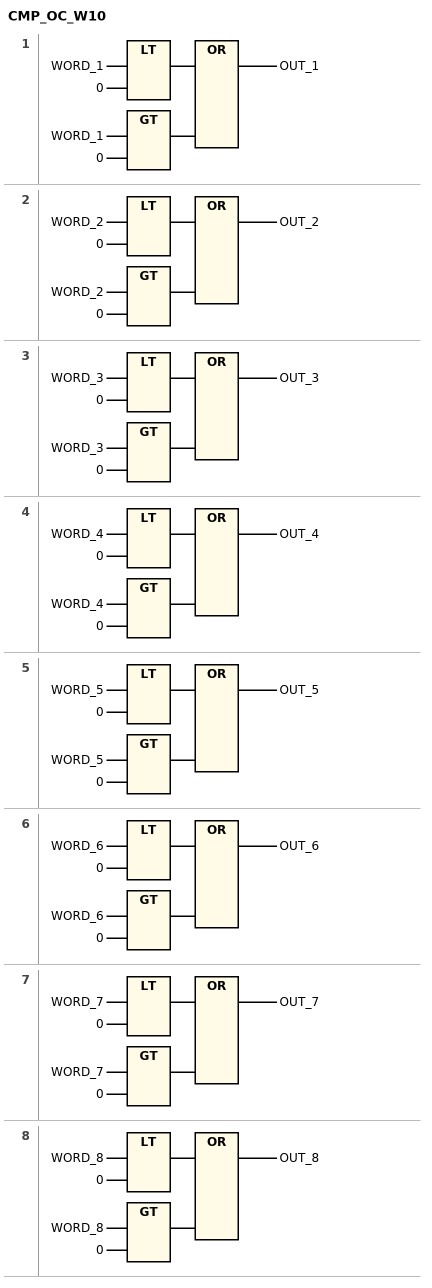
// NETWORK 1
OUT_1 := WORD_1 < 0 OR WORD_1 > 0;

// NETWORK 2
OUT_2 := WORD_2 < 0 OR WORD_2 > 0;

// NETWORK 3
OUT_3 := WORD_3 < 0 OR WORD_3 > 0;

// NETWORK 4
OUT_4 := WORD_4 < 0 OR WORD_4 > 0;

// NETWORK 5
OUT_5 := WORD_5 < 0 OR WORD_5 > 0;

// NETWORK 6
OUT_6 := WORD_6 < 0 OR WORD_6 > 0;

// NETWORK 7
OUT_7 := WORD_7 < 0 OR WORD_7 > 0;

// NETWORK 8
OUT_8 := WORD_8 < 0 OR WORD_8 > 0;

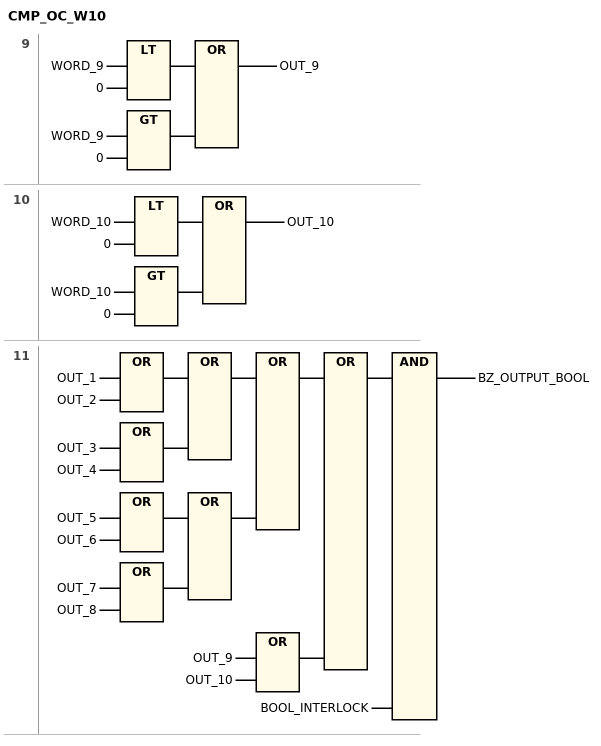
// NETWORK 9
OUT_9 := WORD_9 < 0 OR WORD_9 > 0;

// NETWORK 10
OUT_10 := WORD_10 < 0 OR WORD_10 > 0;

// NETWORK 11
BZ_OUTPUT_BOOL := ((((OUT_1 OR OUT_2) OR (OUT_3 OR OUT_4)) OR ((OUT_5 OR OUT_6) OR (OUT_7 OR OUT_8))) OR (OUT_9 OR OUT_10)) AND BOOL_INTERLOCK;

END_FUNCTION_BLOCK

// ---- FBs/B_JKS_OldFB/Word to Bit/CMP_OC_W2.TcPOU
FUNCTION_BLOCK CMP_OC_W2

VAR_INPUT
	BOOL_INTERLOCK : BOOL; (*INTERLOCK*)
	WORD_1: WORD;		(*WORD 1*)
	WORD_2: WORD;		(*WORD 2*)
	END_VAR


VAR_OUTPUT
	BZ_OUTPUT_BOOL : BOOL;
END_VAR


VAR
	OUT_1: BOOL;
	OUT_2: BOOL;
END_VAR

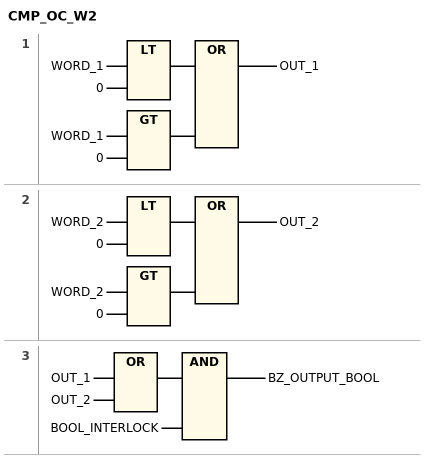
// NETWORK 1
OUT_1 := WORD_1 < 0 OR WORD_1 > 0;

// NETWORK 2
OUT_2 := WORD_2 < 0 OR WORD_2 > 0;

// NETWORK 3
BZ_OUTPUT_BOOL := (OUT_1 OR OUT_2) AND BOOL_INTERLOCK;

END_FUNCTION_BLOCK

// ---- FBs/B_JKS_OldFB/Word to Bit/CMP_OC_W3.TcPOU
FUNCTION_BLOCK CMP_OC_W3

VAR_INPUT
	BOOL_INTERLOCK : BOOL; (*INTERLOCK*)
	WORD_1: WORD;		(*WORD 1*)
	WORD_2: WORD;		(*WORD 2*)
	WORD_3: WORD;		(*WORD 3*)
	END_VAR


VAR_OUTPUT
	BZ_OUTPUT_BOOL : BOOL;
END_VAR


VAR
	OUT_1: BOOL;
	OUT_2: BOOL;
	OUT_3: BOOL;
END_VAR

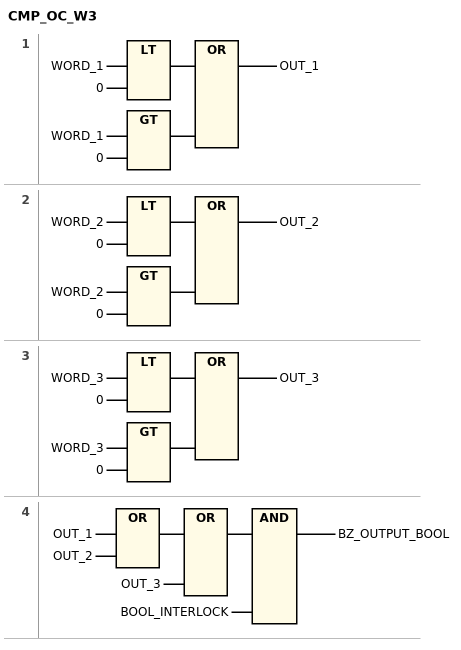
// NETWORK 1
OUT_1 := WORD_1 < 0 OR WORD_1 > 0;

// NETWORK 2
OUT_2 := WORD_2 < 0 OR WORD_2 > 0;

// NETWORK 3
OUT_3 := WORD_3 < 0 OR WORD_3 > 0;

// NETWORK 4
BZ_OUTPUT_BOOL := ((OUT_1 OR OUT_2) OR OUT_3) AND BOOL_INTERLOCK;

END_FUNCTION_BLOCK

// ---- FBs/B_JKS_OldFB/Word to Bit/CMP_OC_W4.TcPOU
FUNCTION_BLOCK CMP_OC_W4

VAR_INPUT
	BOOL_INTERLOCK : BOOL; (*INTERLOCK*)
	WORD_1: WORD;		(*WORD 1*)
	WORD_2: WORD;		(*WORD 2*)
	WORD_3: WORD;		(*WORD 3*)
	WORD_4: WORD;		(*WORD 4*)
	END_VAR


VAR_OUTPUT
	BZ_OUTPUT_BOOL : BOOL;
END_VAR


VAR
	OUT_1: BOOL;
	OUT_2: BOOL;
	OUT_3: BOOL;
	OUT_4: BOOL;
END_VAR

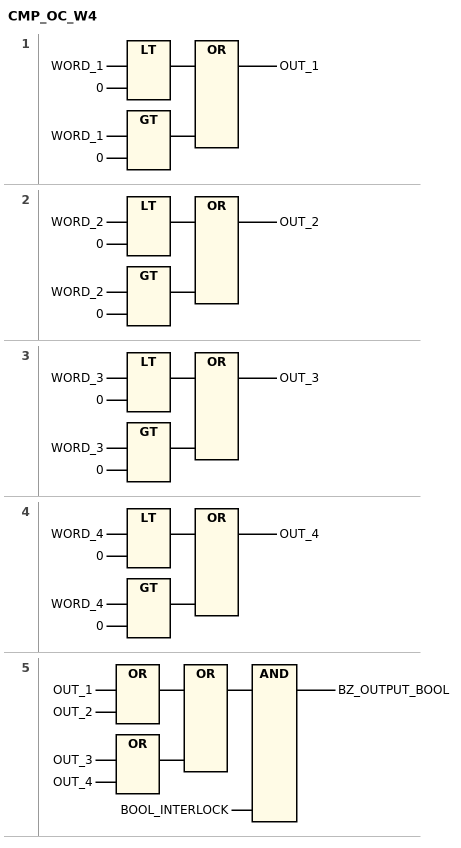
// NETWORK 1
OUT_1 := WORD_1 < 0 OR WORD_1 > 0;

// NETWORK 2
OUT_2 := WORD_2 < 0 OR WORD_2 > 0;

// NETWORK 3
OUT_3 := WORD_3 < 0 OR WORD_3 > 0;

// NETWORK 4
OUT_4 := WORD_4 < 0 OR WORD_4 > 0;

// NETWORK 5
BZ_OUTPUT_BOOL := ((OUT_1 OR OUT_2) OR (OUT_3 OR OUT_4)) AND BOOL_INTERLOCK;

END_FUNCTION_BLOCK

// ---- FBs/B_JKS_OldFB/Word to Bit/CMP_OC_W5.TcPOU
FUNCTION_BLOCK CMP_OC_W5

VAR_INPUT
	BOOL_INTERLOCK : BOOL; (*INTERLOCK*)
	WORD_1: WORD;		(*WORD 1*)
	WORD_2: WORD;		(*WORD 2*)
	WORD_3: WORD;		(*WORD 3*)
	WORD_4: WORD;		(*WORD 4*)
	WORD_5: WORD;		(*WORD 5*)
END_VAR


VAR_OUTPUT
	BZ_OUTPUT_BOOL : BOOL;
END_VAR


VAR
	OUT_1: BOOL;
	OUT_2: BOOL;
	OUT_3: BOOL;
	OUT_4: BOOL;
	OUT_5: BOOL;
END_VAR

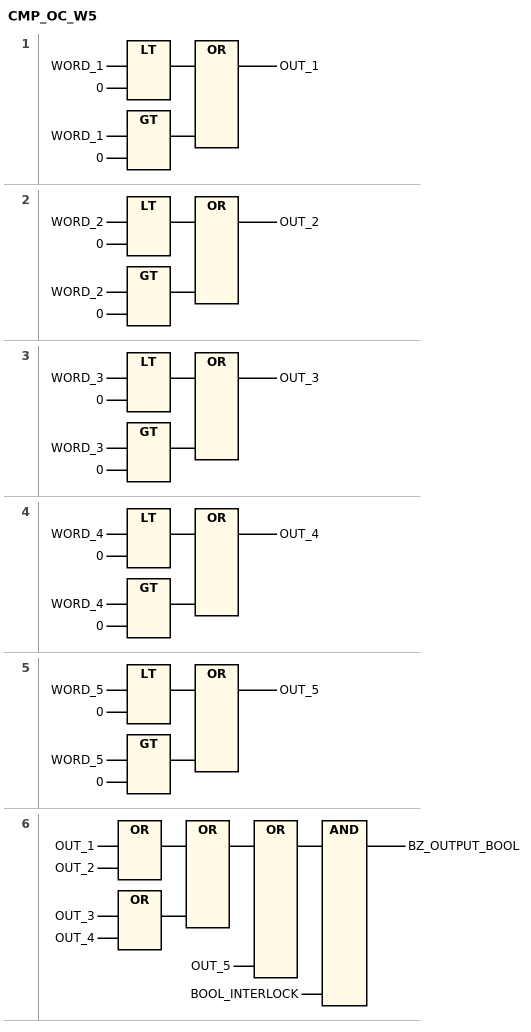
// NETWORK 1
OUT_1 := WORD_1 < 0 OR WORD_1 > 0;

// NETWORK 2
OUT_2 := WORD_2 < 0 OR WORD_2 > 0;

// NETWORK 3
OUT_3 := WORD_3 < 0 OR WORD_3 > 0;

// NETWORK 4
OUT_4 := WORD_4 < 0 OR WORD_4 > 0;

// NETWORK 5
OUT_5 := WORD_5 < 0 OR WORD_5 > 0;

// NETWORK 6
BZ_OUTPUT_BOOL := (((OUT_1 OR OUT_2) OR (OUT_3 OR OUT_4)) OR OUT_5) AND BOOL_INTERLOCK;

END_FUNCTION_BLOCK

// ---- FBs/B_JKS_OldFB/Word to Bit/CMP_OC_W6.TcPOU
FUNCTION_BLOCK CMP_OC_W6

VAR_INPUT
	BOOL_INTERLOCK : BOOL; (*INTERLOCK*)
	WORD_1: WORD;		(*WORD 1*)
	WORD_2: WORD;		(*WORD 2*)
	WORD_3: WORD;		(*WORD 3*)
	WORD_4: WORD;		(*WORD 4*)
	WORD_5: WORD;		(*WORD 5*)
	WORD_6: WORD;		(*WORD 6*)
END_VAR


VAR_OUTPUT
	BZ_OUTPUT_BOOL : BOOL;
END_VAR


VAR
	OUT_1: BOOL;
	OUT_2: BOOL;
	OUT_3: BOOL;
	OUT_4: BOOL;
	OUT_5: BOOL;
	OUT_6: BOOL;
END_VAR

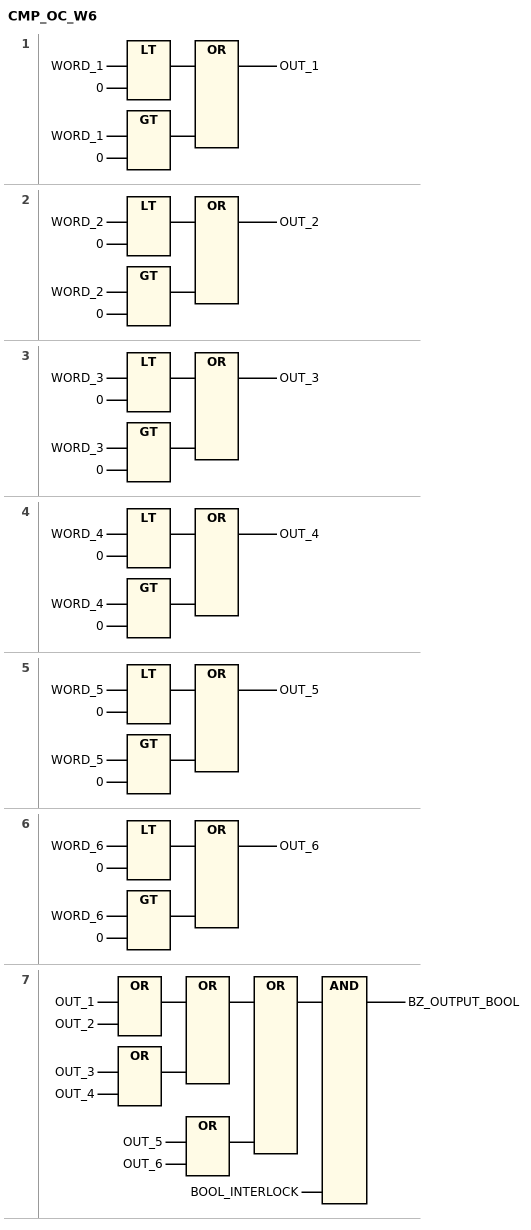
// NETWORK 1
OUT_1 := WORD_1 < 0 OR WORD_1 > 0;

// NETWORK 2
OUT_2 := WORD_2 < 0 OR WORD_2 > 0;

// NETWORK 3
OUT_3 := WORD_3 < 0 OR WORD_3 > 0;

// NETWORK 4
OUT_4 := WORD_4 < 0 OR WORD_4 > 0;

// NETWORK 5
OUT_5 := WORD_5 < 0 OR WORD_5 > 0;

// NETWORK 6
OUT_6 := WORD_6 < 0 OR WORD_6 > 0;

// NETWORK 7
BZ_OUTPUT_BOOL := (((OUT_1 OR OUT_2) OR (OUT_3 OR OUT_4)) OR (OUT_5 OR OUT_6)) AND BOOL_INTERLOCK;

END_FUNCTION_BLOCK

// ---- FBs/B_JKS_OldFB/Word to Bit/CMP_OC_W7.TcPOU
FUNCTION_BLOCK CMP_OC_W7

VAR_INPUT
	BOOL_INTERLOCK : BOOL; (*INTERLOCK*)
	WORD_1: WORD;		(*WORD 1*)
	WORD_2: WORD;		(*WORD 2*)
	WORD_3: WORD;		(*WORD 3*)
	WORD_4: WORD;		(*WORD 4*)
	WORD_5: WORD;		(*WORD 5*)
	WORD_6: WORD;		(*WORD 6*)
	WORD_7: WORD;		(*WORD 7*)
END_VAR


VAR_OUTPUT
	BZ_OUTPUT_BOOL : BOOL;
END_VAR


VAR
	OUT_1: BOOL;
	OUT_2: BOOL;
	OUT_3: BOOL;
	OUT_4: BOOL;
	OUT_5: BOOL;
	OUT_6: BOOL;
	OUT_7: BOOL;
END_VAR

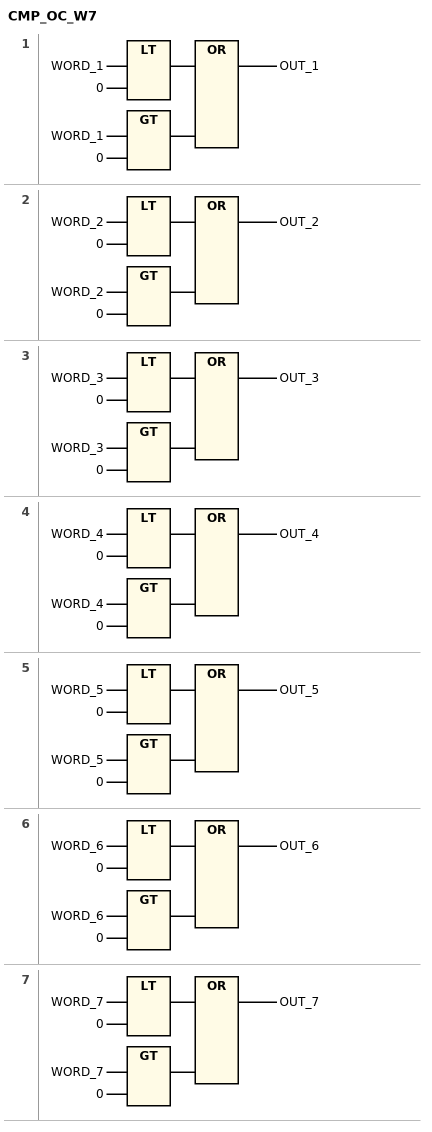
// NETWORK 1
OUT_1 := WORD_1 < 0 OR WORD_1 > 0;

// NETWORK 2
OUT_2 := WORD_2 < 0 OR WORD_2 > 0;

// NETWORK 3
OUT_3 := WORD_3 < 0 OR WORD_3 > 0;

// NETWORK 4
OUT_4 := WORD_4 < 0 OR WORD_4 > 0;

// NETWORK 5
OUT_5 := WORD_5 < 0 OR WORD_5 > 0;

// NETWORK 6
OUT_6 := WORD_6 < 0 OR WORD_6 > 0;

// NETWORK 7
OUT_7 := WORD_7 < 0 OR WORD_7 > 0;

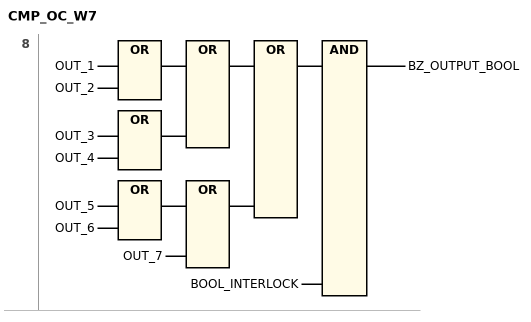
// NETWORK 8
BZ_OUTPUT_BOOL := (((OUT_1 OR OUT_2) OR (OUT_3 OR OUT_4)) OR ((OUT_5 OR OUT_6) OR OUT_7)) AND BOOL_INTERLOCK;

END_FUNCTION_BLOCK

// ---- FBs/B_JKS_OldFB/Word to Bit/CMP_OC_W8.TcPOU
FUNCTION_BLOCK CMP_OC_W8

VAR_INPUT
	BOOL_INTERLOCK : BOOL; (*INTERLOCK*)
	WORD_1: WORD;		(*WORD 1*)
	WORD_2: WORD;		(*WORD 2*)
	WORD_3: WORD;		(*WORD 3*)
	WORD_4: WORD;		(*WORD 4*)
	WORD_5: WORD;		(*WORD 5*)
	WORD_6: WORD;		(*WORD 6*)
	WORD_7: WORD;		(*WORD 7*)
	WORD_8: WORD;		(*WORD 8*)
END_VAR


VAR_OUTPUT
	BZ_OUTPUT_BOOL : BOOL;
END_VAR


VAR
	OUT_1: BOOL;
	OUT_2: BOOL;
	OUT_3: BOOL;
	OUT_4: BOOL;
	OUT_5: BOOL;
	OUT_6: BOOL;
	OUT_7: BOOL;
	OUT_8: BOOL;
END_VAR

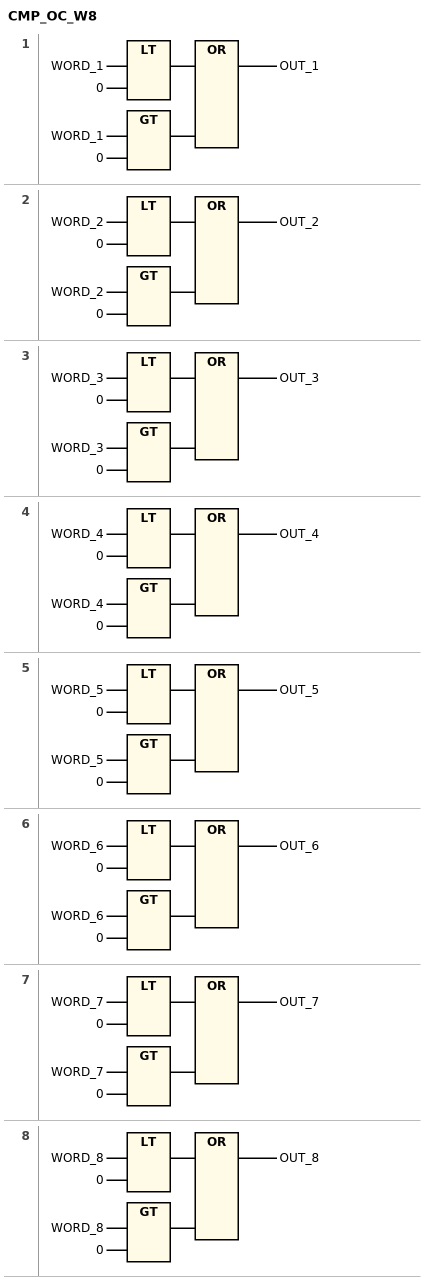
// NETWORK 1
OUT_1 := WORD_1 < 0 OR WORD_1 > 0;

// NETWORK 2
OUT_2 := WORD_2 < 0 OR WORD_2 > 0;

// NETWORK 3
OUT_3 := WORD_3 < 0 OR WORD_3 > 0;

// NETWORK 4
OUT_4 := WORD_4 < 0 OR WORD_4 > 0;

// NETWORK 5
OUT_5 := WORD_5 < 0 OR WORD_5 > 0;

// NETWORK 6
OUT_6 := WORD_6 < 0 OR WORD_6 > 0;

// NETWORK 7
OUT_7 := WORD_7 < 0 OR WORD_7 > 0;

// NETWORK 8
OUT_8 := WORD_8 < 0 OR WORD_8 > 0;

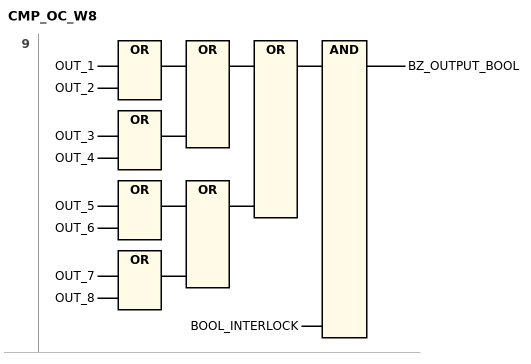
// NETWORK 9
BZ_OUTPUT_BOOL := (((OUT_1 OR OUT_2) OR (OUT_3 OR OUT_4)) OR ((OUT_5 OR OUT_6) OR (OUT_7 OR OUT_8))) AND BOOL_INTERLOCK;

END_FUNCTION_BLOCK

// ---- FBs/B_JKS_OldFB/Word to Bit/CMP_OC_W9.TcPOU
FUNCTION_BLOCK CMP_OC_W9

VAR_INPUT
	BOOL_INTERLOCK : BOOL; (*INTERLOCK*)
	WORD_1: WORD;		(*WORD 1*)
	WORD_2: WORD;		(*WORD 2*)
	WORD_3: WORD;		(*WORD 3*)
	WORD_4: WORD;		(*WORD 4*)
	WORD_5: WORD;		(*WORD 5*)
	WORD_6: WORD;		(*WORD 6*)
	WORD_7: WORD;		(*WORD 7*)
	WORD_8: WORD;		(*WORD 8*)
	WORD_9: WORD;		(*WORD 9*)
END_VAR


VAR_OUTPUT
	BZ_OUTPUT_BOOL : BOOL;
END_VAR


VAR
	OUT_1: BOOL;
	OUT_2: BOOL;
	OUT_3: BOOL;
	OUT_4: BOOL;
	OUT_5: BOOL;
	OUT_6: BOOL;
	OUT_7: BOOL;
	OUT_8: BOOL;
	OUT_9: BOOL;
END_VAR

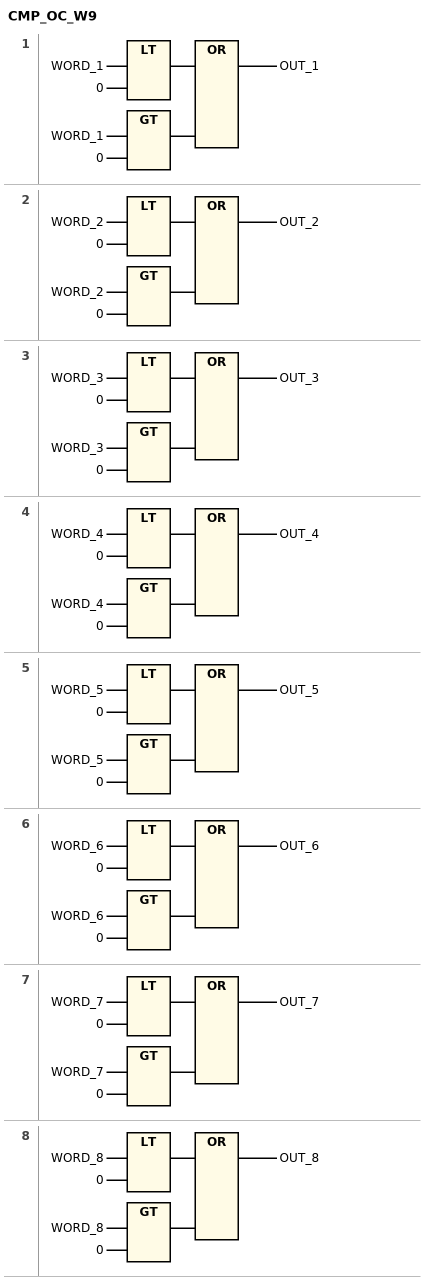
// NETWORK 1
OUT_1 := WORD_1 < 0 OR WORD_1 > 0;

// NETWORK 2
OUT_2 := WORD_2 < 0 OR WORD_2 > 0;

// NETWORK 3
OUT_3 := WORD_3 < 0 OR WORD_3 > 0;

// NETWORK 4
OUT_4 := WORD_4 < 0 OR WORD_4 > 0;

// NETWORK 5
OUT_5 := WORD_5 < 0 OR WORD_5 > 0;

// NETWORK 6
OUT_6 := WORD_6 < 0 OR WORD_6 > 0;

// NETWORK 7
OUT_7 := WORD_7 < 0 OR WORD_7 > 0;

// NETWORK 8
OUT_8 := WORD_8 < 0 OR WORD_8 > 0;

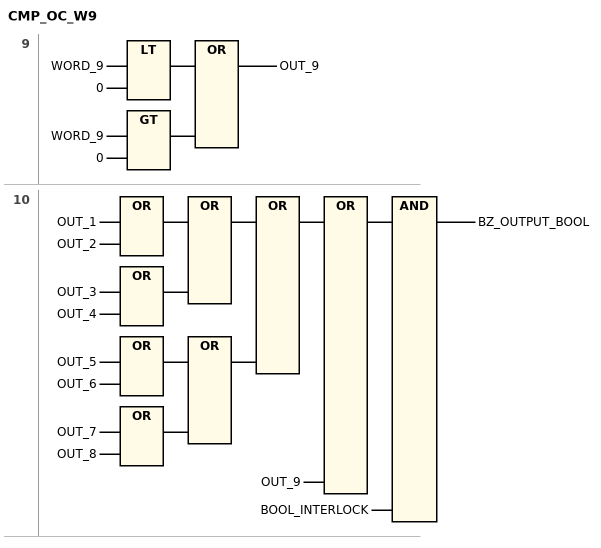
// NETWORK 9
OUT_9 := WORD_9 < 0 OR WORD_9 > 0;

// NETWORK 10
BZ_OUTPUT_BOOL := ((((OUT_1 OR OUT_2) OR (OUT_3 OR OUT_4)) OR ((OUT_5 OR OUT_6) OR (OUT_7 OR OUT_8))) OR OUT_9) AND BOOL_INTERLOCK;

END_FUNCTION_BLOCK

// ---- FBs/FB_Others TBD/fbChemicalMixingWithoutPump.TcPOU
FUNCTION_BLOCK fbChemicalMixingWithoutPump
VAR_INPUT
	bPreparation_Mode	: BOOL;
	bAutoStart_Mode		: BOOL;
	bBasketCounterIN		: BOOL;

	bProTankLowLvl		: BOOL;
	bSubTankLowLvl		: BOOL;
	bSubTankMedLvl		: BOOL;
	bSubTankHighLvl		: BOOL;

END_VAR
VAR_OUTPUT
	bFillingValveOn		: BOOL;
	bPumpOn			: BOOL;
END_VAR
VAR_IN_OUT

	DS_ChemicalMixingTank	: DSChemicalWithoutDosingPump;

END_VAR

VAR PERSISTENT
	iBasketCounter: INT;
END_VAR
VAR
	i1stFill: INT;
	iAutoMode: INT;

	T_MixingTimer: TON;

	R_AutoMode: R_TRIG;
	R_ResetMode: R_TRIG;
	R_1stFill: R_TRIG;
	R_CounterAdd: R_TRIG;
	R_1stFill_1: R_TRIG;
	bChemical1stFillDone: BOOL;
END_VAR

T_MixingTimer(IN:=i1stFill=4 , PT:=DINT_TO_TIME((DS_ChemicalMixingTank.IN_diMixingTime*1000)) , Q=> , ET=> );

R_1stFill(CLK:=bPreparation_Mode  AND NOT bSubTankLowLvl  AND NOT bSubTankMedLvl AND NOT DS_ChemicalMixingTank.OUT_b1stFillCompleted AND NOT bChemical1stFillDone   , Q=> );
R_1stFill_1(CLK:=bPreparation_Mode  AND bSubTankLowLvl  (*AND NOT bSubTankMedLvl*) , Q=> );
R_AutoMode(CLK:=bPreparation_Mode AND bAutoStart_Mode AND bSubTankLowLvl  AND bSubTankMedLvl AND NOT DS_ChemicalMixingTank.IN_bBasketResetQty AND DS_ChemicalMixingTank.OUT_b1stFillCompleted   , Q=> );
R_ResetMode(CLK:=DS_ChemicalMixingTank.IN_bBasketResetQty (*OR  (DS_ChemicalMixingTank.OUT_b1stLimitBasketAlarm OR DS_ChemicalMixingTank.OUT_b2ndLimitBasketAlarm)*)   , Q=> );
R_CounterAdd(CLK:=bAutoStart_Mode AND bBasketCounterIN , Q=> );


DS_ChemicalMixingTank.OUT_iCurrentBasketQty := iBasketCounter ;

IF R_AutoMode.Q THEN
	i1stFill :=6;
END_IF

IF R_ResetMode.Q THEN
iBasketCounter := 0;
END_IF

IF R_1stFill.Q THEN
	i1stFill := 1;
END_IF

IF bSubTankHighLvl THEN
	i1stFill := 5;
END_IF


IF NOT bPreparation_Mode AND NOT bAutoStart_Mode THEN
	i1stFill := 99;
END_IF


IF R_1stFill_1.Q THEN
	i1stFill := 3;
END_IF

CASE i1stFill OF

0:;

1:
	bFillingValveOn := TRUE;

	IF bProTankLowLvl AND bSubTankLowLvl AND NOT bSubTankMedLvl AND NOT bChemical1stFillDone THEN
		i1stFill := 2;
	END_IF

2:
	bFillingValveOn := FALSE;
	DS_ChemicalMixingTank.OUT_b1stFillChemicalTopUpBit := TRUE;

	IF DS_ChemicalMixingTank.IN_bChemicalTopUpNotice THEN
		bChemical1stFillDone	:= TRUE;
		i1stFill := 3;
	END_IF

3:
	DS_ChemicalMixingTank.OUT_b1stFillChemicalTopUpBit := FALSE;

	IF NOT bSubTankMedLvl THEN
		bFillingValveOn := TRUE;
	ELSE
		i1stFill := 4;
	END_IF

4:
	bFillingValveOn := FALSE;
	bPumpOn := TRUE;

	IF T_MixingTimer.Q THEN
		i1stFill := 5;
	END_IF


5:
	DS_ChemicalMixingTank.OUT_b1stFillCompleted := TRUE;
	bPumpOn := FALSE;
	bFillingValveOn := FALSE;
	DS_ChemicalMixingTank.OUT_b1stFillChemicalTopUpBit := FALSE;

	i1stFill := 0;

7:

	i1stFill := 0;


99:
	bFillingValveOn := FALSE;
	bPumpOn := FALSE;
	DS_ChemicalMixingTank.OUT_b1stFillChemicalTopUpBit := FALSE;
	DS_ChemicalMixingTank.OUT_b1stFillCompleted := FALSE;
	bChemical1stFillDone	:= FALSE;

END_CASE

	IF R_CounterAdd.Q THEN
		iBasketCounter := iBasketCounter + 1;
	END_IF

	IF iBasketCounter > DS_ChemicalMixingTank.IN_i1stLimitBasketQty THEN
		DS_ChemicalMixingTank.OUT_b1stLimitBasketAlarm := TRUE;
	END_IF

	IF iBasketCounter > DS_ChemicalMixingTank.IN_i2ndLimitBasketQty THEN
		DS_ChemicalMixingTank.OUT_b2ndLimitBasketAlarm := TRUE;
	END_IF

	IF iBasketCounter <= 0 THEN
		DS_ChemicalMixingTank.OUT_b1stLimitBasketAlarm := FALSE;
		DS_ChemicalMixingTank.OUT_b2ndLimitBasketAlarm := FALSE;
	END_IF

END_FUNCTION_BLOCK

// ---- FBs/FB_Others TBD/fbDetergent_BasketQuantityResetPB_PasswordControl.TcPOU
FUNCTION_BLOCK fbDetergent_BasketQuantityResetPB_PasswordControl
VAR_INPUT
	UserPassword	: ARRAY [0..7] OF STRING;

END_VAR
VAR_IN_OUT
	ARiManualDetergentResetPassword 	: ARRAY [0..iStnQty] OF STRING;

END_VAR

VAR_OUTPUT
	ARbManualDetergentResetFlag			: ARRAY [0..iStnQty] OF BOOL;

END_VAR
VAR
	iSearchFL: INT;
	iCheckFL: INT;
	bResetTriggerFlag: BOOL;
	bResetTriggerTimer: TON;
	ARbManualDetergentResetFlagEmpty			: ARRAY [0..iStnQty] OF BOOL;

END_VAR

iSearchFL := 1;

	FOR iSearchFL := 1 TO iStnQty DO
		IF iSearchFL >= 1 AND iSearchFL <= iStnQty THEN
			IF ARiManualDetergentResetPassword[iSearchFL] <> 'N/A' AND ARiManualDetergentResetPassword[iSearchFL] <> '' THEN
				iCheckFL := 1;
					FOR iCheckFL := 2 TO 7 DO
						IF iCheckFL >= 2 AND iCheckFL <= 7 THEN
							IF ARiManualDetergentResetPassword[iSearchFL] = UserPassword[iCheckFL] THEN
								ARbManualDetergentResetFlag[iSearchFL] := TRUE;
								bResetTriggerFlag := TRUE;
							END_IF
						END_IF
					END_FOR
			END_IF
			ARiManualDetergentResetPassword[iSearchFL] := '';
		END_IF
	END_FOR

bResetTriggerTimer(IN:=bResetTriggerFlag , PT:=t#1s , Q=> , ET=> );

IF bResetTriggerTimer.Q THEN
ARbManualDetergentResetFlag := ARbManualDetergentResetFlagEmpty;
bResetTriggerFlag := FALSE;
END_IF

END_FUNCTION_BLOCK

// ---- FBs/FB_Others TBD/fbMapMobbusTCP.TcPOU
FUNCTION_BLOCK fbMapMobbusTCP
VAR_INPUT

	bEnable					: BOOL;
	sIPAddr					: STRING;
	nMBAddr				: WORD;
	bWriteOut				: ARRAY [0..255] OF BOOL;
	wWriteOut				: ARRAY [0..255] OF WORD;


END_VAR
VAR_OUTPUT

	bReadIn				: ARRAY [0..255] OF BOOL;
	wReadIn					: ARRAY  [0..255] OF WORD;

END_VAR

VAR

	fbWriteCoils				: FB_MBWriteCoils;
	bWriteCoils					: BOOL;

	fbWriteRegs   			: FB_MBWriteRegs;
 	bWriteRegs    			: BOOL;

	fbWriteRegs2   			: FB_MBWriteRegs;
 	bWriteRegs2    			: BOOL;

	fbReadInputRegs     		: FB_MBReadInputRegs;
          bReadRegs       			: BOOL;

	fbReadInputs     			: FB_MBReadInputs;
	 bReadInputs     			: BOOL;

	n						: INT;
	x						: INT;
	start						: BOOL:=TRUE;

	BRead					: ARRAY [0..31] OF BYTE;
	BWrite					: ARRAY [0..31] OF BYTE;
	wWrite					: ARRAY  [0..128] OF WORD;
	wWrite2					: ARRAY  [0..128] OF WORD;




END_VAR

IF bEnable THEN

(*Read Byte/Bool Slave Input coils*)
IF NOT bReadInputs THEN

	 bReadInputs :=TRUE;

	fbReadInputs.sIPAddr		:=sIPAddr;
	fbReadInputs.nQuantity 	:= 256;
	fbReadInputs.nMBAddr 	:= nMBAddr; (*16#8000*)
	fbReadInputs.cbLength 	:= SIZEOF(BRead);
	fbReadInputs.pDestAddr 	:= ADR(BRead);
	fbReadInputs.tTimeout 		:= T#5s;
	fbReadInputs(bExecute:=TRUE);
ELSE
	 IF NOT fbReadInputs.bBUSY THEN
		 bReadInputs:=FALSE;
	END_IF
		 fbReadInputs(bExecute:=FALSE);
END_IF


(*Write Byte/Bool slave Output_coils*)
IF NOT bWriteCoils THEN

	bWriteCoils := TRUE;

	fbWriteCoils.sIPAddr	:=sIPAddr;
	fbWriteCoils.nQuantity 	:=256;
	fbWriteCoils.nMBAddr  := nMBAddr;(*16#8000*)
	fbWriteCoils.cbLength 	:= SIZEOF(BWrite);
	fbWriteCoils.pSrcAddr 	:= ADR(BWrite);
	fbWriteCoils.tTimeout 	:= T#5s;
	fbWriteCoils(bExecute:=TRUE);


ELSE
	IF  NOT fbWriteCoils.bBUSY  THEN
		bWriteCoils :=FALSE;
	END_IF
	fbWriteCoils(bExecute:=FALSE);

END_IF


(*Read word slave  Input_register FB*)
IF NOT bReadRegs THEN

	 bReadRegs :=TRUE;

	 fbReadInputRegs.sIPAddr		:=sIPAddr;
	 fbReadInputRegs.nQuantity		:= 256;
	 fbReadInputRegs.nMBAddr 	:= nMBAddr;(*16#8000*)
	 fbReadInputRegs.cbLength 	:= SIZEOF(wReadIn);
	 fbReadInputRegs.pDestAddr 	:= ADR(wReadIn);
	 fbReadInputRegs.tTimeout 		:= T#5s;
	 fbReadInputRegs(bExecute:=TRUE);
ELSE
	 IF NOT fbReadInputRegs.bBUSY THEN
		 bReadRegs :=FALSE;
	END_IF
		 fbReadInputRegs(bExecute:=FALSE);
END_IF


(* Write Word slave Output_Register (0-128)*)
IF NOT bWriteRegs THEN

	 bWriteRegs :=TRUE;

	 fbWriteRegs.sIPAddr 		:=sIPAddr;
	 fbWriteRegs.nQuantity 		:= 128;
	 fbWriteRegs.nMBAddr 	:= nMBAddr;(*16#8000*)
	 fbWriteRegs.cbLength 		:= SIZEOF(wWrite);
	 fbWriteRegs.pSrcAddr 	:= ADR(wWrite);
	 fbWriteRegs.tTimeout 		:= T#5s;
	 fbWriteRegs(bExecute:=TRUE);

ELSE
	 IF NOT fbWriteRegs.bBUSY THEN
		 bWriteRegs :=FALSE;
	END_IF
		 fbWriteRegs(bExecute:=FALSE);
END_IF


(*Write Word slave Output_Register (129-256)*)
IF NOT bWriteRegs2 THEN

	 bWriteRegs2 :=TRUE;

	 fbWriteRegs2.sIPAddr 		:=sIPAddr;
	 fbWriteRegs2.nQuantity	:= 128;
	 fbWriteRegs2.nMBAddr 	:=(nMBAddr+16#0080); (*16#8080 is 128*)
	 fbWriteRegs2.cbLength 	:= SIZEOF(wWrite2);
	 fbWriteRegs2.pSrcAddr 	:= ADR(wWrite2);
	 fbWriteRegs2.tTimeout 	:= T#5s;
	 fbWriteRegs2(bExecute:=TRUE);

ELSE
	 IF NOT fbWriteRegs2.bBUSY THEN
		 bWriteRegs2 :=FALSE;
	END_IF
		 fbWriteRegs2(bExecute:=FALSE);
END_IF


(* Write register word from two FB variables to one variable*)
IF start THEN
	FOR
		n:=0 TO 128 DO

			wWrite[n]:=wWriteOut[n];

	END_FOR

	x:=0;
	FOR
		n:=128 TO 255 DO
	
			wWrite2[x]:=wWriteOut[n];
			x:=x+1;
	END_FOR

END_IF







(* Write Bool to Byte Mapping*)
		BWrite[0].0:=bWriteOut[0];
		BWrite[0].1:=BWriteOut[1];
		BWrite[0].2:=BWriteOut[2];
		BWrite[0].3:=BWriteOut[3];
		BWrite[0].4:=BWriteOut[4];
		BWrite[0].5:=BWriteOut[5];
		BWrite[0].6:=BWriteOut[6];
		BWrite[0].7:=BWriteOut[7];

		BWrite[1].0:=BWriteOut[8];
		BWrite[1].1:=BWriteOut[9];
		BWrite[1].2:=BWriteOut[10];
		BWrite[1].3:=BWriteOut[11];
		BWrite[1].4:=BWriteOut[12];
		BWrite[1].5:=BWriteOut[13];
		BWrite[1].6:=BWriteOut[14];
		BWrite[1].7:=BWriteOut[15];

		BWrite[2].0:=BWriteOut[16];
		BWrite[2].1:=BWriteOut[17];
		BWrite[2].2:=BWriteOut[18];
		BWrite[2].3:=BWriteOut[19];
		BWrite[2].4:=BWriteOut[20];
		BWrite[2].5:=BWriteOut[21];
		BWrite[2].6:=BWriteOut[22];
		BWrite[2].7:=BWriteOut[23];

		BWrite[3].0:=BWriteOut[24];
		BWrite[3].1:=BWriteOut[25];
		BWrite[3].2:=BWriteOut[26];
		BWrite[3].3:=BWriteOut[27];
		BWrite[3].4:=BWriteOut[28];
		BWrite[3].5:=BWriteOut[29];
		BWrite[3].6:=BWriteOut[30];
		BWrite[3].7:=BWriteOut[31];

		BWrite[4].0:=BWriteOut[32];
		BWrite[4].1:=BWriteOut[33];
		BWrite[4].2:=BWriteOut[34];
		BWrite[4].3:=BWriteOut[35];
		BWrite[4].4:=BWriteOut[36];
		BWrite[4].5:=BWriteOut[37];
		BWrite[4].6:=BWriteOut[38];
		BWrite[4].7:=BWriteOut[39];

		BWrite[5].0:=BWriteOut[40];
		BWrite[5].1:=BWriteOut[41];
		BWrite[5].2:=BWriteOut[42];
		BWrite[5].3:=BWriteOut[43];
		BWrite[5].4:=BWriteOut[44];
		BWrite[5].5:=BWriteOut[45];
		BWrite[5].6:=BWriteOut[46];
		BWrite[5].7:=BWriteOut[47];

		BWrite[6].0:=BWriteOut[48];
		BWrite[6].1:=BWriteOut[49];
		BWrite[6].2:=BWriteOut[50];
		BWrite[6].3:=BWriteOut[51];
		BWrite[6].4:=BWriteOut[52];
		BWrite[6].5:=BWriteOut[53];
		BWrite[6].6:=BWriteOut[54];
		BWrite[6].7:=BWriteOut[55];

		BWrite[7].0:=BWriteOut[56];
		BWrite[7].1:=BWriteOut[57];
		BWrite[7].2:=BWriteOut[58];
		BWrite[7].3:=BWriteOut[59];
		BWrite[7].4:=BWriteOut[60];
		BWrite[7].5:=BWriteOut[61];
		BWrite[7].6:=BWriteOut[62];
		BWrite[7].7:=BWriteOut[63];

		BWrite[8].0:=BWriteOut[64];
		BWrite[8].1:=BWriteOut[65];
		BWrite[8].2:=BWriteOut[66];
		BWrite[8].3:=BWriteOut[67];
		BWrite[8].4:=BWriteOut[68];
		BWrite[8].5:=BWriteOut[69];
		BWrite[8].6:=BWriteOut[70];
		BWrite[8].7:=BWriteOut[71];

		BWrite[9].0:=BWriteOut[72];
		BWrite[9].1:=BWriteOut[73];
		BWrite[9].2:=BWriteOut[74];
		BWrite[9].3:=BWriteOut[75];
		BWrite[9].4:=BWriteOut[76];
		BWrite[9].5:=BWriteOut[77];
		BWrite[9].6:=BWriteOut[78];
		BWrite[9].7:=BWriteOut[79];

		BWrite[10].0:=BWriteOut[80];
		BWrite[10].1:=BWriteOut[81];
		BWrite[10].2:=BWriteOut[82];
		BWrite[10].3:=BWriteOut[83];
		BWrite[10].4:=BWriteOut[84];
		BWrite[10].5:=BWriteOut[85];
		BWrite[10].6:=BWriteOut[86];
		BWrite[10].7:=BWriteOut[87];

		BWrite[11].0:=BWriteOut[88];
		BWrite[11].1:=BWriteOut[89];
		BWrite[11].2:=BWriteOut[90];
		BWrite[11].3:=BWriteOut[91];
		BWrite[11].4:=BWriteOut[92];
		BWrite[11].5:=BWriteOut[93];
		BWrite[11].6:=BWriteOut[94];
		BWrite[11].7:=BWriteOut[95];

		BWrite[12].0:=BWriteOut[96];
		BWrite[12].1:=BWriteOut[97];
		BWrite[12].2:=BWriteOut[98];
		BWrite[12].3:=BWriteOut[99];
		BWrite[12].4:=BWriteOut[100];
		BWrite[12].5:=BWriteOut[101];
		BWrite[12].6:=BWriteOut[102];
		BWrite[12].7:=BWriteOut[103];

		BWrite[13].0:=BWriteOut[104];
		BWrite[13].1:=BWriteOut[105];
		BWrite[13].2:=BWriteOut[106];
		BWrite[13].3:=BWriteOut[107];
		BWrite[13].4:=BWriteOut[108];
		BWrite[13].5:=BWriteOut[109];
		BWrite[13].6:=BWriteOut[110];
		BWrite[13].7:=BWriteOut[111];

		BWrite[14].0:=BWriteOut[112];
		BWrite[14].1:=BWriteOut[113];
		BWrite[14].2:=BWriteOut[114];
		BWrite[14].3:=BWriteOut[115];
		BWrite[14].4:=BWriteOut[116];
		BWrite[14].5:=BWriteOut[117];
		BWrite[14].6:=BWriteOut[118];
		BWrite[14].7:=BWriteOut[119];

		BWrite[15].0:=BWriteOut[120];
		BWrite[15].1:=BWriteOut[121];
		BWrite[15].2:=BWriteOut[122];
		BWrite[15].3:=BWriteOut[123];
		BWrite[15].4:=BWriteOut[124];
		BWrite[15].5:=BWriteOut[125];
		BWrite[15].6:=BWriteOut[126];
		BWrite[15].7:=BWriteOut[127];

		BWrite[16].0:=BWriteOut[128];
		BWrite[16].1:=BWriteOut[129];
		BWrite[16].2:=BWriteOut[130];
		BWrite[16].3:=BWriteOut[131];
		BWrite[16].4:=BWriteOut[132];
		BWrite[16].5:=BWriteOut[133];
		BWrite[16].6:=BWriteOut[134];
		BWrite[16].7:=BWriteOut[135];

		BWrite[17].0:=BWriteOut[136];
		BWrite[17].1:=BWriteOut[137];
		BWrite[17].2:=BWriteOut[138];
		BWrite[17].3:=BWriteOut[139];
		BWrite[17].4:=BWriteOut[140];
		BWrite[17].5:=BWriteOut[141];
		BWrite[17].6:=BWriteOut[142];
		BWrite[17].7:=BWriteOut[143];

		BWrite[18].0:=BWriteOut[144];
		BWrite[18].1:=BWriteOut[145];
		BWrite[18].2:=BWriteOut[146];
		BWrite[18].3:=BWriteOut[147];
		BWrite[18].4:=BWriteOut[148];
		BWrite[18].5:=BWriteOut[149];
		BWrite[18].6:=BWriteOut[150];
		BWrite[18].7:=BWriteOut[151];

		BWrite[19].0:=BWriteOut[152];
		BWrite[19].1:=BWriteOut[153];
		BWrite[19].2:=BWriteOut[154];
		BWrite[19].3:=BWriteOut[155];
		BWrite[19].4:=BWriteOut[156];
		BWrite[19].5:=BWriteOut[157];
		BWrite[19].6:=BWriteOut[158];
		BWrite[19].7:=BWriteOut[159];

		BWrite[20].0:=BWriteOut[160];
		BWrite[20].1:=BWriteOut[161];
		BWrite[20].2:=BWriteOut[162];
		BWrite[20].3:=BWriteOut[163];
		BWrite[20].4:=BWriteOut[164];
		BWrite[20].5:=BWriteOut[165];
		BWrite[20].6:=BWriteOut[166];
		BWrite[20].7:=BWriteOut[167];
		BWrite[21].0:=BWriteOut[168];

		BWrite[21].1:=BWriteOut[169];
		BWrite[21].2:=BWriteOut[170];
		BWrite[21].3:=BWriteOut[171];
		BWrite[21].4:=BWriteOut[172];
		BWrite[21].5:=BWriteOut[173];
		BWrite[21].6:=BWriteOut[174];
		BWrite[21].7:=BWriteOut[175];

		BWrite[22].0:=BWriteOut[176];
		BWrite[22].1:=BWriteOut[177];
		BWrite[22].2:=BWriteOut[178];
		BWrite[22].3:=BWriteOut[179];
		BWrite[22].4:=BWriteOut[180];
		BWrite[22].5:=BWriteOut[181];
		BWrite[22].6:=BWriteOut[182];
		BWrite[22].7:=BWriteOut[183];

		BWrite[23].0:=BWriteOut[184];
		BWrite[23].1:=BWriteOut[185];
		BWrite[23].2:=BWriteOut[186];
		BWrite[23].3:=BWriteOut[187];
		BWrite[23].4:=BWriteOut[188];
		BWrite[23].5:=BWriteOut[189];
		BWrite[23].6:=BWriteOut[190];
		BWrite[23].7:=BWriteOut[191];

		BWrite[24].0:=BWriteOut[192];
		BWrite[24].1:=BWriteOut[193];
		BWrite[24].2:=BWriteOut[194];
		BWrite[24].3:=BWriteOut[195];
		BWrite[24].4:=BWriteOut[196];
		BWrite[24].5:=BWriteOut[197];
		BWrite[24].6:=BWriteOut[198];
		BWrite[24].7:=BWriteOut[199];

		BWrite[25].0:=BWriteOut[200];
		BWrite[25].1:=BWriteOut[201];
		BWrite[25].2:=BWriteOut[202];
		BWrite[25].3:=BWriteOut[203];
		BWrite[25].4:=BWriteOut[204];
		BWrite[25].5:=BWriteOut[205];
		BWrite[25].6:=BWriteOut[206];
		BWrite[25].7:=BWriteOut[207];

		BWrite[26].0:=BWriteOut[208];
		BWrite[26].1:=BWriteOut[209];
		BWrite[26].2:=BWriteOut[210];
		BWrite[26].3:=BWriteOut[211];
		BWrite[26].4:=BWriteOut[212];
		BWrite[26].5:=BWriteOut[213];
		BWrite[26].6:=BWriteOut[214];
		BWrite[26].7:=BWriteOut[215];

		BWrite[27].0:=BWriteOut[216];
		BWrite[27].1:=BWriteOut[217];
		BWrite[27].2:=BWriteOut[218];
		BWrite[27].3:=BWriteOut[219];
		BWrite[27].4:=BWriteOut[220];
		BWrite[27].5:=BWriteOut[221];
		BWrite[27].6:=BWriteOut[222];
		BWrite[27].7:=BWriteOut[223];

		BWrite[28].0:=BWriteOut[224];
		BWrite[28].1:=BWriteOut[225];
		BWrite[28].2:=BWriteOut[226];
		BWrite[28].3:=BWriteOut[227];
		BWrite[28].4:=BWriteOut[228];
		BWrite[28].5:=BWriteOut[229];
		BWrite[28].6:=BWriteOut[230];
		BWrite[28].7:=BWriteOut[231];

		BWrite[29].0:=BWriteOut[232];
		BWrite[29].1:=BWriteOut[233];
		BWrite[29].2:=BWriteOut[234];
		BWrite[29].3:=BWriteOut[235];
		BWrite[29].4:=BWriteOut[236];
		BWrite[29].5:=BWriteOut[237];
		BWrite[29].6:=BWriteOut[238];
		BWrite[29].7:=BWriteOut[239];

		BWrite[30].0:=BWriteOut[240];
		BWrite[30].1:=BWriteOut[241];
		BWrite[30].2:=BWriteOut[242];
		BWrite[30].3:=BWriteOut[243];
		BWrite[30].4:=BWriteOut[244];
		BWrite[30].5:=BWriteOut[245];
		BWrite[30].6:=BWriteOut[246];
		BWrite[30].7:=BWriteOut[247];

		BWrite[30].0:=BWriteOut[248];
		BWrite[31].1:=BWriteOut[249];
		BWrite[31].2:=BWriteOut[250];
		BWrite[31].3:=BWriteOut[251];
		BWrite[31].4:=BWriteOut[252];
		BWrite[31].5:=BWriteOut[253];
		BWrite[31].6:=BWriteOut[254];
		BWrite[31].7:=BWriteOut[255];



		(*Read Byte to Bool mapping*)
		bReadIn[0]:=BRead[0].0;
		bReadIn[1]:=BRead[0].1;
		bReadIn[2]:=BRead[0].2;
		bReadIn[3]:=BRead[0].3;
		bReadIn[4]:=BRead[0].4;
		bReadIn[5]:=BRead[0].5;
		bReadIn[6]:=BRead[0].6;
		bReadIn[7]:=BRead[0].7;

		bReadIn[8]:=BRead[1].0;
		bReadIn[9]:=BRead[1].1;
		bReadIn[10]:=BRead[1].2;
		bReadIn[11]:=BRead[1].3;
		bReadIn[12]:=BRead[1].4;
		bReadIn[13]:=BRead[1].5;
		bReadIn[14]:=BRead[1].6;
		bReadIn[15]:=BRead[1].7;

		bReadIn[16]:=BRead[2].0;
		bReadIn[17]:=BRead[2].1;
		bReadIn[18]:=BRead[2].2;
		bReadIn[19]:=BRead[2].3;
		bReadIn[20]:=BRead[2].4;
		bReadIn[21]:=BRead[2].5;
		bReadIn[22]:=BRead[2].6;
		bReadIn[23]:=BRead[2].7;

		bReadIn[24]:=BRead[3].0;
		bReadIn[25]:=BRead[3].1;
		bReadIn[26]:=BRead[3].2;
		bReadIn[27]:=BRead[3].3;
		bReadIn[28]:=BRead[3].4;
		bReadIn[29]:=BRead[3].5;
		bReadIn[30]:=BRead[3].6;
		bReadIn[31]:=BRead[3].7;

		bReadIn[32]:=BRead[4].0;
		bReadIn[33]:=BRead[4].1;
		bReadIn[34]:=BRead[4].2;
		bReadIn[35]:=BRead[4].3;
		bReadIn[36]:=BRead[4].4;
		bReadIn[37]:=BRead[4].5;
		bReadIn[38]:=BRead[4].6;
		bReadIn[39]:=BRead[4].7;

		bReadIn[40]:=BRead[5].0;
		bReadIn[41]:=BRead[5].1;
		bReadIn[42]:=BRead[5].2;
		bReadIn[43]:=BRead[5].3;
		bReadIn[44]:=BRead[5].4;
		bReadIn[45]:=BRead[5].5;
		bReadIn[46]:=BRead[5].6;
		bReadIn[47]:=BRead[5].7;

		bReadIn[48]:=BRead[6].0;
		bReadIn[49]:=BRead[6].1;
		bReadIn[50]:=BRead[6].2;
		bReadIn[51]:=BRead[6].3;
		bReadIn[52]:=BRead[6].4;
		bReadIn[53]:=BRead[6].5;
		bReadIn[54]:=BRead[6].6;
		bReadIn[55]:=BRead[6].7;

		bReadIn[56]:=BRead[7].0;
		bReadIn[57]:=BRead[7].1;
		bReadIn[58]:=BRead[7].2;
		bReadIn[59]:=BRead[7].3;
		bReadIn[60]:=BRead[7].4;
		bReadIn[61]:=BRead[7].5;
		bReadIn[62]:=BRead[7].6;
		bReadIn[63]:=BRead[7].7;

		bReadIn[64]:=BRead[8].0;
		bReadIn[65]:=BRead[8].1;
		bReadIn[66]:=BRead[8].2;
		bReadIn[67]:=BRead[8].3;
		bReadIn[68]:=BRead[8].4;
		bReadIn[69]:=BRead[8].5;
		bReadIn[70]:=BRead[8].6;
		bReadIn[71]:=BRead[8].7;

		bReadIn[72]:=BRead[9].0;
		bReadIn[73]:=BRead[9].1;
		bReadIn[74]:=BRead[9].2;
		bReadIn[75]:=BRead[9].3;
		bReadIn[76]:=BRead[9].4;
		bReadIn[77]:=BRead[9].5;
		bReadIn[78]:=BRead[9].6;
		bReadIn[79]:=BRead[9].7;

		bReadIn[80]:=BRead[10].0;
		bReadIn[81]:=BRead[10].1;
		bReadIn[82]:=BRead[10].2;
		bReadIn[83]:=BRead[10].3;
		bReadIn[84]:=BRead[10].4;
		bReadIn[85]:=BRead[10].5;
		bReadIn[86]:=BRead[10].6;
		bReadIn[87]:=BRead[10].7;

		bReadIn[88]:=BRead[11].0;
		bReadIn[89]:=BRead[11].1;
		bReadIn[90]:=BRead[11].2;
		bReadIn[91]:=BRead[11].3;
		bReadIn[92]:=BRead[11].4;
		bReadIn[93]:=BRead[11].5;
		bReadIn[94]:=BRead[11].6;
		bReadIn[95]:=BRead[11].7;

		bReadIn[96]:=BRead[12].0;
		bReadIn[97]:=BRead[12].1;
		bReadIn[98]:=BRead[12].2;
		bReadIn[99]:=BRead[12].3;
		bReadIn[100]:=BRead[12].4;
		bReadIn[101]:=BRead[12].5;
		bReadIn[102]:=BRead[12].6;
		bReadIn[103]:=BRead[12].7;

		bReadIn[104]:=BRead[13].0;
		bReadIn[105]:=BRead[13].1;
		bReadIn[106]:=BRead[13].2;
		bReadIn[107]:=BRead[13].3;
		bReadIn[108]:=BRead[13].4;
		bReadIn[109]:=BRead[13].5;
		bReadIn[110]:=BRead[13].6;
		bReadIn[111]:=BRead[13].7;

		bReadIn[112]:=BRead[14].0;
		bReadIn[113]:=BRead[14].1;
		bReadIn[114]:=BRead[14].2;
		bReadIn[115]:=BRead[14].3;
		bReadIn[116]:=BRead[14].4;
		bReadIn[117]:=BRead[14].5;
		bReadIn[118]:=BRead[14].6;
		bReadIn[119]:=BRead[14].7;

		bReadIn[120]:=BRead[15].0;
		bReadIn[121]:=BRead[15].1;
		bReadIn[122]:=BRead[15].2;
		bReadIn[123]:=BRead[15].3;
		bReadIn[124]:=BRead[15].4;
		bReadIn[125]:=BRead[15].5;
		bReadIn[126]:=BRead[15].6;
		bReadIn[127]:=BRead[15].7;

		bReadIn[128]:=BRead[16].0;
		bReadIn[129]:=BRead[16].1;
		bReadIn[130]:=BRead[16].2;
		bReadIn[131]:=BRead[16].3;
		bReadIn[132]:=BRead[16].4;
		bReadIn[133]:=BRead[16].5;
		bReadIn[134]:=BRead[16].6;
		bReadIn[135]:=BRead[16].7;

		bReadIn[136]:=BRead[17].0;
		bReadIn[137]:=BRead[17].1;
		bReadIn[138]:=BRead[17].2;
		bReadIn[139]:=BRead[17].3;
		bReadIn[140]:=BRead[17].4;
		bReadIn[141]:=BRead[17].5;
		bReadIn[142]:=BRead[17].6;
		bReadIn[143]:=BRead[17].7;

		bReadIn[144]:=BRead[18].0;
		bReadIn[145]:=BRead[18].1;
		bReadIn[146]:=BRead[18].2;
		bReadIn[147]:=BRead[18].3;
		bReadIn[148]:=BRead[18].4;
		bReadIn[149]:=BRead[18].5;
		bReadIn[150]:=BRead[18].6;
		bReadIn[151]:=BRead[18].7;

		bReadIn[152]:=BRead[19].0;
		bReadIn[153]:=BRead[19].1;
		bReadIn[154]:=BRead[19].2;
		bReadIn[155]:=BRead[19].3;
		bReadIn[156]:=BRead[19].4;
		bReadIn[157]:=BRead[19].5;
		bReadIn[158]:=BRead[19].6;
		bReadIn[159]:=BRead[19].7;

		bReadIn[160]:=BRead[20].0;
		bReadIn[161]:=BRead[20].1;
		bReadIn[162]:=BRead[20].2;
		bReadIn[163]:=BRead[20].3;
		bReadIn[164]:=BRead[20].4;
		bReadIn[165]:=BRead[20].5;
		bReadIn[166]:=BRead[20].6;
		bReadIn[167]:=BRead[20].7;

		bReadIn[168]:=BRead[21].0;
		bReadIn[169]:=BRead[21].1;
		bReadIn[170]:=BRead[21].2;
		bReadIn[171]:=BRead[21].3;
		bReadIn[172]:=BRead[21].4;
		bReadIn[173]:=BRead[21].5;
		bReadIn[174]:=BRead[21].6;
		bReadIn[175]:=BRead[21].7;

		bReadIn[176]:=BRead[22].0;
		bReadIn[177]:=BRead[22].1;
		bReadIn[178]:=BRead[22].2;
		bReadIn[179]:=BRead[22].3;
		bReadIn[180]:=BRead[22].4;
		bReadIn[181]:=BRead[22].5;
		bReadIn[182]:=BRead[22].6;
		bReadIn[183]:=BRead[22].7;

		bReadIn[184]:=BRead[23].0;
		bReadIn[185]:=BRead[23].1;
		bReadIn[186]:=BRead[23].2;
		bReadIn[187]:=BRead[23].3;
		bReadIn[188]:=BRead[23].4;
		bReadIn[189]:=BRead[23].5;
		bReadIn[190]:=BRead[23].6;
		bReadIn[191]:=BRead[23].7;

		bReadIn[192]:=BRead[24].0;
		bReadIn[193]:=BRead[24].1;
		bReadIn[194]:=BRead[24].2;
		bReadIn[195]:=BRead[24].3;
		bReadIn[196]:=BRead[24].4;
		bReadIn[197]:=BRead[24].5;
		bReadIn[198]:=BRead[24].6;
		bReadIn[199]:=BRead[24].7;

		bReadIn[200]:=BRead[25].0;
		bReadIn[201]:=BRead[25].1;
		bReadIn[202]:=BRead[25].2;
		bReadIn[203]:=BRead[25].3;
		bReadIn[204]:=BRead[25].4;
		bReadIn[205]:=BRead[25].5;
		bReadIn[206]:=BRead[25].6;
		bReadIn[207]:=BRead[25].7;

		bReadIn[208]:=BRead[26].0;
		bReadIn[209]:=BRead[26].1;
		bReadIn[210]:=BRead[26].2;
		bReadIn[211]:=BRead[26].3;
		bReadIn[212]:=BRead[26].4;
		bReadIn[213]:=BRead[26].5;
		bReadIn[214]:=BRead[26].6;
		bReadIn[215]:=BRead[26].7;

		bReadIn[216]:=BRead[27].0;
		bReadIn[217]:=BRead[27].1;
		bReadIn[218]:=BRead[27].2;
		bReadIn[219]:=BRead[27].3;
		bReadIn[220]:=BRead[27].4;
		bReadIn[221]:=BRead[27].5;
		bReadIn[222]:=BRead[27].6;
		bReadIn[223]:=BRead[27].7;

		bReadIn[224]:=BRead[28].0;
		bReadIn[225]:=BRead[28].1;
		bReadIn[226]:=BRead[28].2;
		bReadIn[227]:=BRead[28].3;
		bReadIn[228]:=BRead[28].4;
		bReadIn[229]:=BRead[28].5;
		bReadIn[230]:=BRead[28].6;
		bReadIn[231]:=BRead[28].7;

		bReadIn[232]:=BRead[29].0;
		bReadIn[233]:=BRead[29].1;
		bReadIn[234]:=BRead[29].2;
		bReadIn[235]:=BRead[29].3;
		bReadIn[236]:=BRead[29].4;
		bReadIn[237]:=BRead[29].5;
		bReadIn[238]:=BRead[29].6;
		bReadIn[239]:=BRead[29].7;

		bReadIn[240]:=BRead[30].0;
		bReadIn[241]:=BRead[30].1;
		bReadIn[242]:=BRead[30].2;
		bReadIn[243]:=BRead[30].3;
		bReadIn[244]:=BRead[30].4;
		bReadIn[245]:=BRead[30].5;
		bReadIn[246]:=BRead[30].6;
		bReadIn[247]:=BRead[30].7;
		bReadIn[248]:=BRead[30].0;

		bReadIn[249]:=BRead[31].1;
		bReadIn[250]:=BRead[31].2;
		bReadIn[251]:=BRead[31].3;
		bReadIn[252]:=BRead[31].4;
		bReadIn[253]:=BRead[31].5;
		bReadIn[254]:=BRead[31].6;
		bReadIn[255]:=BRead[31].7;




END_IF

END_FUNCTION_BLOCK

// ---- FBs/FB_Others TBD/fbOilSeperatorTankCtrl.TcPOU
FUNCTION_BLOCK fbOilSeperatorTankCtrl
VAR_INPUT
	bEnable			: BOOL;
	bOilLowLevel		: BOOL;
	bOilHighLevel	: BOOL;
	bResetCounter	: BOOL;
	iDrainCounterSV	: INT;
END_VAR
VAR_OUTPUT
	bDrainingValve	: BOOL;
	bOilTankFull		: BOOL;

END_VAR
VAR_OUTPUT PERSISTENT
	iDrainCounterPV	: INT;
END_VAR

VAR
	T_HighLevel: TON;

	F_LowLevel: F_TRIG;
	R_CounterAdd: R_TRIG;
END_VAR

IF bEnable THEN

T_HighLevel(IN:=bOilHighLevel , PT:=T#3S , Q=> , ET=> );
F_LowLevel(CLK:=bOilLowLevel , Q=> );
R_CounterAdd(CLK:=bDrainingValve , Q=> );

	IF bOilLowLevel AND bOilHighLevel AND T_HighLevel.Q THEN
		bDrainingValve := TRUE;
	END_IF

	IF F_LowLevel.Q THEN
		bDrainingValve := FALSE;
	END_IF

	IF R_CounterAdd.Q THEN
		iDrainCounterPV := iDrainCounterPV +1;
	END_IF

	IF iDrainCounterPV >= iDrainCounterSV THEN
		bOilTankFull := TRUE;
	ELSE
		bOilTankFull := FALSE;
	END_IF

	IF bResetCounter THEN
		iDrainCounterPV := 0;
	END_IF

ELSE

	bDrainingValve := FALSE;

END_IF

END_FUNCTION_BLOCK

// ---- FBs/FB_Others TBD/fbV3_LoadingRecipeCheck.TcPOU
FUNCTION_BLOCK fbV3_LoadingRecipeCheck
VAR_INPUT

	iLoadingRecipeNo : INT;
	ARsProductRecipeDescription: ARRAY [0..iProductRecipeArrayQty] OF STRING(50);

END_VAR
VAR_OUTPUT

	bRecipeAvailable : BOOL;
	bRecipeNotAvailable : BOOL;
END_VAR
VAR
END_VAR


	IF iLoadingRecipeNo > 0 THEN

		IF ARsProductRecipeDescription[iLoadingRecipeNo] = '' THEN
		bRecipeNotAvailable := TRUE;
		bRecipeAvailable := FALSE;
		ELSE
		bRecipeNotAvailable := FALSE;
		bRecipeAvailable := TRUE;
		END_IF

	ELSE

		bRecipeNotAvailable := FALSE;
		bRecipeAvailable := FALSE;

	END_IF

END_FUNCTION_BLOCK

// ---- FBs/FB_Others TBD/PID_FB.TcPOU
FUNCTION_BLOCK PID_FB
VAR_INPUT
	fSetpointValue_INT			: INT						;
	PID_fKp						: REAL (*:= 1.0	*)				;
	PID_tTn						: TIME (*:= T#1s*)				;
	PID_tTv						: TIME (*:= T#30ms*)				;
	PID_tTd						: TIME (*:= T#40ms	*)			;

END_VAR

VAR_IN_OUT
	fActualValueINT		: INT				;	(*this is the measured value. you need to map this variable to the hardware input*)
END_VAR
VAR_OUTPUT
	fOutREAL_INT AT %Q*			: INT				;	(*this is the output value. you need to map this variable to the hardware output*)
	iOutPercent					: INT				;
END_VAR


VAR
	fSetpointValue				: FLOAT				; 	(*this is your set point value*)

	fActualValue					: FLOAT				;
	fActualValueINT_REAL			:REAL				;

	fOut 							: FLOAT				;
	bHold						: BOOL				;

	fManSyncValue				: FLOAT				;
	bSync						: BOOL				;


	eMode						: E_CTRL_MODE		;
	stCTRL_PID_PARAMS			: ST_CTRL_PID_PARAMS;

	eErrorId					: E_CTRL_ERRORCODES;
	bError						: BOOL				;
	bARWactive					: BOOL				;

	(* controller *)
	fbCTRL_PID					: FB_CTRL_PID		;

	bInit							: BOOL	:= TRUE		;
	fbTON						: TON				;

	fSetpointValueToScope		: FLOAT				;
	fActualValueToScope			: FLOAT				;
	fOutToScope					: FLOAT				;

END_VAR

;IF bInit
THEN
	(* init parameter struct *)
	stCTRL_PID_PARAMS.tCtrlCycleTime		:= T#10ms;
	stCTRL_PID_PARAMS.tTaskCycleTime		:= T#10ms;
	stCTRL_PID_PARAMS.fKp					:= PID_fKp;			(* proportional gain Kp*)
	stCTRL_PID_PARAMS.tTn					:= PID_tTn;			(*  Tn *)
	stCTRL_PID_PARAMS.tTv					:= PID_tTv;		(*  Tv *)
	stCTRL_PID_PARAMS.tTd					:= PID_tTd;		(*  Td *)
	stCTRL_PID_PARAMS.fOutMaxLimit			:=  100;			(* maximum output limit	*)
	stCTRL_PID_PARAMS.fOutMinLimit			:= 0;			(* minimum output limit	*)

	(* set the mode to ACTIVE --> normal operation *)
	eMode							:= eCTRL_MODE_ACTIVE;

	(* reset the init flag *)
	bInit							:= FALSE;
END_IF

fSetpointValue:=INT_TO_FLOAT(fSetpointValue_INT);

(*fActualValueINT_REAL:=INT_TO_REAL(fActualValueINT);
fActualValueINT_REAL:=fActualValueINT_REAL*10/32767;*)
fActualValue:=INT_TO_FLOAT(fActualValueINT);

fOutREAL_INT:=FLOAT_TO_INT(fOut*327.67);
iOutPercent:=FLOAT_TO_INT(fOut);
(*fOutREAL_INT:=fOutREAL_INT*32767/100;*)

fSetpointValueToScope 	:= fSetpointValue;
fActualValueToScope 		:= fActualValue;

(* call controller *)
fbCTRL_PID(			fSetpointValue		:= fSetpointValue,
					fActualValue			:= fActualValue,
					fManSyncValue		:= fManSyncValue,
					bSync				:= bSync,
					eMode				:= eMode,
					bHold				:= bHold,
					stParams			:= stCTRL_PID_PARAMS,
					fOut					=> fOut,
					bARWactive			=> bARWactive,
					eErrorId				=> eErrorId,
					bError				=> bError
				);
(* copy var to scope var *)
fOutToScope := fOutREAL_INT;

END_FUNCTION_BLOCK

// ---- POUs/MainProgram/CheckBound/CheckBounds.TcPOU
FUNCTION CheckBounds :DINT
VAR_INPUT
	index, lower, upper 	:DINT;
END_VAR
VAR
END_VAR

IF index<lower THEN
	CheckBounds_ErrCnt := CheckBounds_ErrCnt + 1;
	CheckBounds := lower;
ELSIF index>upper THEN
	CheckBounds_ErrCnt := CheckBounds_ErrCnt + 1;
	CheckBounds := upper;
ELSE
	CheckBounds := index;
END_IF

END_FUNCTION

// ---- POUs/MainProgram/CheckBound/CheckDivByte.TcPOU
FUNCTION CheckDivByte : BYTE
VAR_INPUT
	divisor			 	: BYTE;
END_VAR
VAR
END_VAR

IF divisor = 0 THEN
	CheckByteZeroDiv_ErrCnt := CheckByteZeroDiv_ErrCnt + 1;
	CheckDivByte := 1;
ELSE
	CheckDivByte := divisor;
END_IF

END_FUNCTION

// ---- POUs/MainProgram/CheckBound/CheckDivDWord.TcPOU
FUNCTION CheckDivDWord : DWORD
VAR_INPUT
	divisor				: DWORD;
END_VAR
VAR
END_VAR

IF divisor = 0 THEN
	CheckDWordZeroDiv_ErrCnt := CheckDWordZeroDiv_ErrCnt + 1;
	CheckDivDWord := 1;
ELSE
	CheckDivDWord := divisor;
END_IF

END_FUNCTION

// ---- POUs/MainProgram/CheckBound/CheckDivLreal.TcPOU
FUNCTION CheckDivLreal : LREAL
VAR_INPUT
	divisor		 		: LREAL;
END_VAR
VAR
END_VAR

IF divisor = 0 THEN
	CheckLrealZeroDiv_ErrCnt := CheckLrealZeroDiv_ErrCnt + 1;
	CheckDivLreal := 1;
ELSE
	CheckDivLreal := divisor;
END_IF

END_FUNCTION

// ---- POUs/MainProgram/CheckBound/CheckDivReal.TcPOU
FUNCTION CheckDivReal : REAL
VAR_INPUT
	divisor		 		: REAL;
END_VAR
VAR
END_VAR

IF divisor = 0 THEN
	CheckRealZeroDiv_ErrCnt := CheckRealZeroDiv_ErrCnt + 1;
	CheckDivReal := 1;
ELSE
	CheckDivReal := divisor;
END_IF

END_FUNCTION

// ---- POUs/MainProgram/CheckBound/CheckRangeSigned.TcPOU
FUNCTION CheckRangeSigned : DINT
VAR_INPUT
	value, lower, upper 	: DINT;
END_VAR
VAR
END_VAR

IF value<lower THEN
	CheckRangeSigned_ErrCnt := CheckRangeSigned_ErrCnt + 1;
	CheckRangeSigned := lower;
ELSIF value>upper THEN
	CheckRangeSigned_ErrCnt := CheckRangeSigned_ErrCnt + 1;
	CheckRangeSigned := upper;
ELSE
	CheckRangeSigned := value;
END_IF

END_FUNCTION

// ---- POUs/MainProgram/Other/HMI_Invinsible_Ctrl.TcPOU
PROGRAM HMI_Invinsible_Ctrl
VAR
	x: BOOL;
	y: BOOL;
END_VAR

//1
IF NOT Global_HMI.bManualOutToUserConfirmPageOn THEN 
	Global_HMI.bManualOutToUserConfirmPageOff:=TRUE;
ELSE
	Global_HMI.bManualOutToUserConfirmPageOff:=FALSE;
END_IF

//2
IF NOT Global_Variables_HMI_Function.bStationOnPage THEN
	Global_Variables_HMI_Function.bStationOffPage :=TRUE;
ELSE
	Global_Variables_HMI_Function.bStationOffPage :=FALSE;
END_IF

//3
IF NOT Global_Variables_HMI_Function.RecipeEditOn THEN
	Global_Variables_HMI_Function.RecipeEditOff :=TRUE;
ELSE
	Global_Variables_HMI_Function.RecipeEditOff :=FALSE;
END_IF

//4
IF NOT NOT Global_HMI.bManualOutToUserConfirmPageOn THEN
	Global_HMI.bManualOutToUserConfirmPageOff :=TRUE;
ELSE
	Global_HMI.bManualOutToUserConfirmPageOff :=FALSE;
END_IF

//5
IF NOT x THEN
	y :=TRUE;
ELSE
	y :=FALSE;
END_IF

//6
IF NOT x THEN
	y :=TRUE;
ELSE
	y :=FALSE;
END_IF

//7
IF NOT x THEN
	y :=TRUE;
ELSE
	y :=FALSE;
END_IF

//8
IF NOT x THEN
	y :=TRUE;
ELSE
	y :=FALSE;
END_IF

//9
IF NOT x THEN
	y :=TRUE;
ELSE
	y :=FALSE;
END_IF

//10
IF NOT x THEN
	y :=TRUE;
ELSE
	y :=FALSE;
END_IF

//11
IF NOT x THEN
	y :=TRUE;
ELSE
	y :=FALSE;
END_IF

//12
IF NOT x THEN
	y :=TRUE;
ELSE
	y :=FALSE;
END_IF

//13
IF NOT x THEN
	y :=TRUE;
ELSE
	y :=FALSE;
END_IF

//14
IF NOT x THEN
	y :=TRUE;
ELSE
	y :=FALSE;
END_IF

//15
IF NOT x THEN
	y :=TRUE;
ELSE
	y :=FALSE;
END_IF

END_PROGRAM

// ---- GlobalTextList.TcGTLO
TEXTLIST GlobalTextList
  2681 = '     '
  119 = '%'
  1446 = '%0.01f'
  4503 = '%0.02f'
  2738 = '%0.1f'
  537 = '%d'
  890 = '%i'
  889 = '%s'
  2909 = '(X100.00) STN 01 - 03 ULTRASONIC GENERATOR MCB - TRIP (-10F1)\n'
  3104 = '(X100.01) STN 01 ULTRASONIC GENERATOR (LEFT & RIGHT) - ALARM (-10U1)'
  9404 = '(X100.02) STN 01 ULTRASONIC GENERATOR (BOTTOM) - ALARM (-10U1)\n'
  10481 = '(X100.03) STN 02 ULTRASONIC GENERATOR (LEFT & RIGHT) - ALARM (-10U1)\n'
  10488 = '(X100.04) STN 02 ULTRASONIC GENERATOR (BOTTOM) - ALARM (-10U1)\n'
  5247 = '(X100.05) STN 03 ULTRASONIC GENERATOR (LEFT & RIGHT) - ALARM (-10U1)'
  11591 = '(X100.06) STN 03 ULTRASONIC GENERATOR (BOTTOM) - ALARM (-10U1)'
  12139 = '(X100.07) STN 04 - 05 ULTRASONIC GENERATOR MCB - TRIP (-11F1)'
  6933 = '(X100.08) STN 04 ULTRASONIC GENERATOR (LEFT & RIGHT) - ALARM (-11U1)'
  6619 = '(X100.09) STN 04 ULTRASONIC GENERATOR (BOTTOM) - ALARM (-11U1)'
  4361 = '(X100.10) STN 05 ULTRASONIC GENERATOR (BOTTOM) - ALARM (-11U1)'
  1199 = '(X100.11) GENERAL MAIN PANEL PB - E-STOP (-251S1)'
  10185 = '(X100.12) OPERATOR PULL STRING - E-STOP (-251S2)'
  10087 = '(X100.13) MAINTENANCE PULL STRING - E-STOP  (-251S3)'
  6489 = '(X100.14) GENERAL TOUCH MONITOR SOCKET ELCB - TRIP (-8Q1)'
  7510 = '(X100.15) ARM 01 SERVO DRIVE MCB - TRIP (-40F1)'
  11212 = '(X101.00) IPC DC ON SIGNAL (-410K1)'
  2968 = '(X101.01) PANEL VENTILATION FAN MCB - TRIP  (-6F1)\n'
  9585 = '(X101.02) PANEL LIGHTING MCB - TRIP  (-5F1)'
  4159 = '(X101.03) MACHINE LIGHTING 01 MCB - TRIP (-5F2)'
  7312 = '(X101.04) MACHINE LIGHTING 02 MCB - TRIP (-5F3)'
  4346 = '(X101.05) GENERAL TOUCH MONITOR SOCKET MCB - TRIP (-8F1)'
  8277 = '(X101.06) GENERAL PHASE SEQUENCE RELAY MCB - TRIP (-3F2)'
  9048 = '(X101.07) GENERAL PHASE SEQUENCE RELAY - TRIP (-3K1)'
  10253 = '(X101.08) STN 06 PROCESS TANK BLOWER MMS&TOR - TRIP (-100Q1)'
  5932 = '(X101.09) STN 01 - 06 EXHAUST BLOWER MMS&TOR - TRIP (-101Q1)'
  6620 = '(X101.10) STN 01 - 05 AGITATION MOTOR MMS&TOR - TRIP (-160Q1)'
  5425 = '(X101.11) STN 01 DOSING PUMP MCB - TRIP (-70F1)'
  3137 = '(X101.12) STN 02 DOSING PUMP MCB - TRIP (-71F1)'
  3866 = '(X101.13) STN 03 DOSING PUMP MCB - TRIP (-72F1)'
  11364 = '(X101.14) STN 04 DOSING PUMP MCB - TRIP (-73F1)'
  8857 = '(X101.15) STN 01 DOSING CHEMICAL CONTAINER RELAY SIGNAL - FEEDBACK (-70K1)'
  620 = '(X102.00) STN 01 PROCESS TANK PUMP MMS&TOR - TRIP (-74Q1)'
  9751 = '(X102.01) STN 02 PROCESS TANK PUMP MMS&TOR - TRIP (-75Q1)'
  11969 = '(X102.02) STN 03 PROCESS TANK PUMP MMS&TOR - TRIP (-76Q1)'
  9673 = '(X102.03) STN 04 PROCESS TANK PUMP MMS&TOR - TRIP (-77Q1)'
  4653 = '(X102.04) STN 05 PROCESS TANK PUMP MMS&TOR - TRIP (-78Q1)'
  1689 = '(X102.05) STN 01 - 04 CHEMICAL RETURN TANK PUMP MMS&TOR - TRIP (-80Q1)'
  5529 = '(X102.06) STN 06 PROCESS TANK VACUUM PUMP MMS&TOR -TRIP (-79Q1)'
  315 = '(X102.07) STN 01 PROCESS TANK HEATER MCB - TRIP (-130F1)'
  910 = '(X102.08) STN 02 PROCESS TANK HEATER MCB - TRIP (-131F1)'
  6525 = '(X102.09) STN 03 PROCESS TANK HEATER MCB - TRIP (-132F1)'
  11585 = '(X102.10) STN 04 PROCESS TANK HEATER MCB - TRIP (-133F1)'
  3596 = '(X102.11) STN 06 PROCESS TANK HEATER MCB - TRIP (-134F1)'
  1057 = '(X102.12) LOADING CONVEYOR 1 MCB - TRIP (-170F1)'
  11382 = '(X102.13) LOADING CONVEYOR 2 MCB - TRIP (-171F1)'
  1453 = '(X102.14) LOADING CONVEYOR 3 MCB - TRIP (-172F1)'
  1076 = '(X102.15) STN 02 DOSING CHEMICAL CONTAINER RELAY SIGNAL - FEEDBACK (-71K1)\n'
  2864 = '(X103.00) MAIN SAFETY CONTACTOR 1 - FEEDBACK  (-250K1)'
  3842 = '(X103.01) MAIN SAFETY CONTACTOR 2 - FEEDBACK  (-250K2)'
  9985 = '(X103.02) DOOR SAFETY  CONTACTOR 1 - FEEDBACK  (-255K1)'
  4912 = '(X103.03) DOOR SAFETY  CONTACTOR 2 - FEEDBACK  (-255K2)'
  7342 = '(X103.04) MODULE 01 ADDITIONAL POWER SUPPLY INCOMING POWER MCB -TRIP (-4F3)\n'
  8981 = '(X103.05) MODULE 01 ADDITIONAL POWER SUPPLY OUTGOING POWER MCB -TRIP (-4F4)'
  2731 = '(X103.06) MODULE 02 ADDITIONAL POWER SUPPLY INCOMING POWER MCB -TRIP (-4F5)'
  8822 = '(X103.07) MODULE 02 ADDITIONAL POWER SUPPLY OUTGOING POWER MCB -TRIP (-4F6)'
  6849 = '(X103.08) MODULE 03 ADDITIONAL POWER SUPPLY INCOMING POWER MCB -TRIP (-4F7)'
  3806 = '(X103.09) MODULE 03 ADDITIONAL POWER SUPPLY OUTGOING POWER MCB -TRIP (-4F8)'
  2985 = '(X103.10) ARM 01 ADDITIONAL POWER SUPPLY INCOMING POWER MCB -TRIP (-4F9)'
  4712 = '(X103.11) ARM 01 ADDITIONAL POWER SUPPLY OUTGOING POWER MCB -TRIP (-4F10)'
  7888 = '(X103.12) STN 05 - 06 FFU UNIT MCB - TRIP (-163F1)'
  12134 = '(X103.13) UNLOADING FFU UNIT MCB - TRIP (-164F1)'
  150 = '(X103.14) RESERVED'
  7835 = '(X103.15) RESERVED'
  4580 = '(X104.00) GENERAL ALARM PB - RESET (-304S1)'
  12604 = '(X104.01) GENERAL BUZZER PB - RESET (-304S2)'
  85 = '(X104.02) STN 01 PROCESS TANK SENSOR - MAX O/F (-304B1)'
  2048 = '(X104.03) STN 01 PROCESS TANK SENSOR - MIN O/F (-304B2)'
  9817 = '(X104.04) STN 01 PROCESS TANK SENSOR - MIN (-304B3)'
  527 = '(X104.05) STN 02 PROCESS TANK SENSOR - MAX O/F (-304B4)'
  4696 = '(X104.06) STN 02 PROCESS TANK SENSOR - MIN O/F (-304B5)'
  4065 = '(X104.07) STN 02 PROCESS TANK SENSOR - MIN (-304B6)'
  1186 = '(X104.08) STN 01 DOSING CHEMICAL CONTAINER SENSOR - WARNING LEVEL (-304S3)'
  10163 = '(X104.09) STN 01 DOSING CHEMICAL CONTAINER SENSOR - MIN LEVEL (-304S3)'
  11193 = '(X104.10) STRUCTURE 01 DRIP PAN SENSOR - LEAK (-304B7)'
  12677 = '(X104.11) STN 02 DOSING CHEMICAL CONTAINER SENSOR - WARNING LEVEL (-304S4)'
  10077 = '(X104.12) STN 02 DOSING CHEMICAL CONTAINER SENSOR - MIN LEVEL (-304S4)'
  4208 = '(X104.13) ARM 01 HORIZONTAL SENSOR - LOADING OT (-304B8)'
  2010 = '(X104.14) ARM 01 HORIZONTAL SENSOR - HOME (-304B9)'
  6891 = '(X104.15) GENERAL SAFETY CURTAIN SENSOR - ALARM (-255K3)'
  12989 = '(X110.00) ARM 01 VERTICAL SENSOR - TOP OT (-310B7)'
  10651 = '(X110.01) ARM 01 VERTICAL SENSOR - HOME (-310B8)'
  7995 = '(X110.02) ARM 01 VERTICAL SENSOR - BTM OT (-310B9)'
  9097 = '(X110.03) ARM 01 VERTICAL SENSOR - CRASH (-310B10)'
  4152 = '(X110.04) ARM 01 SENSOR A - MISSHOOK (-310B11)'
  5728 = '(X110.05) ARM 01 SENSOR B - MISSHOOK (-310B12)'
  10051 = '(X110.06) STN 03 PROCESS TANK SENSOR - MAX O/F (-310B1)'
  11634 = '(X110.07) STN 03 PROCESS TANK SENSOR - MIN O/F (-310B2)'
  362 = '(X110.08) STN 03 PROCESS TANK SENSOR - MIN (-310B3)'
  1438 = '(X110.09) STN 04 PROCESS TANK SENSOR - MAX O/F (-310B4)'
  11723 = '(X110.10) STN 04 PROCESS TANK SENSOR - MIN (-310B5)'
  10513 = '(X110.11) STRUCTURE 02 DRIP PAN SENSOR - LEAK (-310B6)'
  11762 = '(X110.12) STN 03 DOSING CHEMICAL CONTAINER SENSOR - WARNING LEVEL (-310S1)\n'
  3924 = '(X110.13) STN 03 DOSING CHEMICAL CONTAINER SENSOR - MIN LEVEL (-310S1)'
  505 = '(X110.14) STN 04 DOSING CHEMICAL CONTAINER SENSOR - WARNING LEVEL (-310S2)'
  11202 = '(X110.15) STN 04 DOSING CHEMICAL CONTAINER SENSOR - MIN LEVEL (-310S2)'
  1533 = '(X111.00) STN 03 DOSING CHEMICAL CONTAINER RELAY SIGNAL - FEEDBACK (-72K1)'
  12520 = '(X111.01) STN 04 DOSING CHEMICAL CONTAINER RELAY SIGNAL - FEEDBACK (-73K1)'
  4899 = '(X111.02) STN 04 PROCESS TANK SENSOR - MIN O/F (-311B1)'
  5642 = '(X111.03) RESERVED\n'
  3322 = '(X111.04) RESERVED'
  421 = '(X111.05) RESERVED'
  1655 = '(X111.06) RESERVED'
  9383 = '(X111.07) RESERVED'
  6156 = '(X111.08) RESERVED'
  9743 = '(X111.09) RESERVED\n'
  5314 = '(X111.10) RESERVED'
  3972 = '(X111.11) RESERVED\n'
  3844 = '(X111.12) RESERVED'
  636 = '(X111.13) RESERVED\n'
  2624 = '(X111.14) RESERVED\n'
  1246 = '(X111.15) RESERVED\n'
  4633 = '(X120.00) STN 05 PROCESS TANK SENSOR - MAX O/F (-320B1)'
  11874 = '(X120.01) STN 05 PROCESS TANK SENSOR - MIN (-320B2)'
  9495 = '(X120.02) STN 01 - 04 CHEMICAL RETURN TANK SENSOR - MAX (-320B3)'
  9155 = '(X120.03) STN 01 - 04 CHEMICAL RETURN TANK SENSOR - REG (-320B4)'
  10251 = '(X120.04) STN 01 - 04 CHEMICAL RETURN TANK SENSOR - MIN (-320B5)'
  1697 = '(X120.05) STN 05 PROCESS TANK FLOW SENSOR - MIN FLOW (-320S1)'
  3762 = '(X120.06) STN 06 PROCESS TANK HEATER THERMOSTAT - ALARM (-320S2)'
  10613 = '(X120.07) STN 06 SHUTTER DOOR RS - OPEN (-320S3)'
  2184 = '(X120.08) STN 06 SHUTTER DOOR RS - CLOSE (-320S4)'
  7879 = '(X120.09) STRUCTURE 03 DRIP PAN SENSOR - LEAK (-320B6)'
  4230 = '(X120.10) GENERAL INCOMING CDA PRESSURE SWITCH - MIN PRESSURE (-320S5)'
  4949 = '(X120.11) UNLOADING SENSOR - BASKET DETECTION (-320B7)'
  12570 = '(X120.12) ARM 01 HORIZONTAL SENSOR - UNLOADING OT (-320B8)'
  3635 = '(X120.13) RESERVED'
  2627 = '(X120.14) RESERVED'
  1145 = '(X120.15) RESERVED'
  7632 = '(X121.00) STN 06 SHUTTER DOOR RS 01 - CLAMP (-321S1)'
  3825 = '(X121.01) STN 06 SHUTTER DOOR RS 01 - UNCLAMP (-321S2)'
  10015 = '(X121.02) STN 06 SHUTTER DOOR RS 02 - CLAMP (-321S3)'
  615 = '(X121.03) STN 06 SHUTTER DOOR RS 02 - UNCLAMP (-321S4)\n'
  10327 = '(X121.04) RESERVED'
  2759 = '(X121.05) RESERVED'
  1035 = '(X121.07) RESERVED\n'
  12534 = '(X121.08) RESERVED\n'
  400 = '(X121.09) RESERVED'
  7041 = '(X121.10) RESERVED\n'
  13024 = '(X121.11) RESERVED'
  6920 = '(X121.12) RESERVED\n'
  2569 = '(X121.13) RESERVED\n'
  1238 = '(X121.14) RESERVED\n'
  4602 = '(X121.15) RESERVED\n'
  12780 = '(X12130.06) RESERVED'
  6575 = '(X130.00) LOADING CONVEYOR SENSOR - FEED (-330B1)'
  4551 = '(X130.01) LOADING CONVEYOR SENSOR - INDEX (-330B2)\n'
  12720 = '(X130.02) LOADING CONVEYOR SENSOR - PICK  (-330B3)'
  10446 = '(X130.03) GENERAL LOADING PB - E-STOP (-251S4)'
  7225 = '(X130.04) RESERVED'
  2132 = '(X130.05) RESERVED\n'
  1761 = '(X130.06) RESERVED\n'
  4766 = '(X130.07) RESERVED'
  1698 = '(X130.08) RESERVED\n'
  3688 = '(X130.09) RESERVED\n'
  7104 = '(X130.10) RESERVED\n'
  1854 = '(X130.11) RESERVED\n'
  5960 = '(X130.12) RESERVED\n'
  4771 = '(X130.13) RESERVED\n'
  185 = '(X130.14) RESERVED\n'
  1144 = '(X130.15) RESERVED\n'
  9162 = '(Y100.00) EMERGENCY STOP SAFETY RELAY - RESET  (-250K3)\\'
  12386 = '(Y100.01) STN 01 - 03 ULTRASONIC GENERATOR FREQUENCY CHANGE BIT 1 (-10U1)'
  9328 = '(Y100.02) STN 01 - 03 ULTRASONIC GENERATOR FREQUENCY CHANGE BIT 2 (-10U1)'
  9208 = '(Y100.03) STN 04 - 05 ULTRASONIC GENERATOR FREQUENCY CHANGE BIT 1 (-11U1)'
  3667 = '(Y100.04) STN 04 - 05 ULTRASONIC GENERATOR FREQUENCY CHANGE BIT 2 (-11U1)'
  4791 = '(Y100.05) GENERAL ALARM RESET IND (-304S1)'
  6872 = '(Y100.06) GENERAL BUZZER  RESET IND (-304S2)'
  1691 = '(Y100.07) GENERAL BUZZER TONE 1 (-400H1)'
  5301 = '(Y100.08) GENERAL BUZZER TONE 2 (-400H1)'
  3358 = '(Y100.09) GENERAL TOWER LIGHT IND - RED (-400H2)'
  7213 = '(Y100.10) GENERAL TOWER LIGHT IND - YELLOW (-400H2)'
  1059 = '(Y100.11) GENERAL TOWER LIGHT IND - GREEN (-400H2)'
  3384 = '(Y100.12) RESERVED(Y100.12) IPC DC ON HOLDING RELAY (-400K1)\n'
  1106 = '(Y100.13) STN 05 - 06 FFU UNIT ON/OFF ()'
  12934 = '(Y100.14) UNLOADING FFU UNIT ON/OFF ()'
  6399 = '(Y100.15) RESERVED\n'
  10014 = '(Y101.00) STN 01 ULTRASONIC GENERATOR (LEFT &RIGHT) ON/OFF (-10U1)'
  9375 = '(Y101.01) STN 01 ULTRASONIC GENERATOR (BOTTOM) ON/OFF (-10U1)'
  739 = '(Y101.02) STN 02 ULTRASONIC GENERATOR (LEFT &RIGHT) ON/OFF (-10U1)'
  12798 = '(Y101.03) STN 02 ULTRASONIC GENERATOR (BOTTOM) ON/OFF (-10U1)'
  12492 = '(Y101.04) STN 03 ULTRASONIC GENERATOR (LEFT &RIGHT) ON/OFF (-10U1)'
  9197 = '(Y101.05) STN 03 ULTRASONIC GENERATOR (BOTTOM) ON/OFF (-10U1)'
  12029 = '(Y101.06) STN 04 ULTRASONIC GENERATOR (LEFT &RIGHT) ON/OFF (-11U1)'
  11238 = '(Y101.07) STN 04 ULTRASONIC GENERATOR (BOTTOM) ON/OFF (-11U1)'
  3974 = '(Y101.08) STN 05 ULTRASONIC GENERATOR (BOTTOM) ON/OFF (-11U1)'
  10864 = '(Y101.09) STN 01 DOSING PUMP ON/OFF (-70K1)'
  2375 = '(Y101.10) STN 02 DOSING PUMP ON/OFF (-71K1)'
  9806 = '(Y101.11) STN 01 PROCESS TANK PUMP ON/OFF (-74K1)'
  11195 = '(Y101.12) STN 02 PROCESS TANK PUMP ON/OFF (-75K1)'
  9429 = '(Y101.13) STN 03 PROCESS TANK PUMP ON/OFF (-76K1)'
  12323 = '(Y101.14) STN 04 PROCESS TANK PUMP ON/OFF (-77K1)'
  13519 = '(Y101.15) STN 05 PROCESS TANK PUMP ON/OFF (-78K1)'
  2957 = '(Y102.00) STN 01 - 04 CHEMICAL RETURN TANK PUMP ON/OFF (-80K1)'
  4102 = '(Y102.01) STN 06 PROCESS TANK VACUUM PUMP ON/OFF (-79K1)'
  7047 = '(Y102.02) STN 01 PROCESS TANK HEATER ON/OFF (-130K1)'
  11795 = '(Y102.03) STN 02 PROCESS TANK HEATER ON/OFF (-131K1)'
  4147 = '(Y102.04) STN 03 PROCESS TANK HEATER ON/OFF (-132K1)'
  1831 = '(Y102.05) STN 04 PROCESS TANK HEATER ON/OFF (-133K1)'
  4645 = '(Y102.06) STN 06 PROCESS TANK HEATER ON/OFF (-134K1)'
  1347 = '(Y102.07) STN 06 PROCESS TANK BLOWER ON/OFF (-100K1)'
  8847 = '(Y102.08) STN 01 - 06 EXHAUST BLOWER ON/OFF (-101K1)'
  11090 = '(Y102.09) RESERVED'
  6826 = '(Y102.10) RESERVED\n'
  9055 = '(Y102.11) RESERVED'
  8987 = '(Y102.12) RESERVED'
  1210 = '(Y102.13) RESERVED'
  7178 = '(Y102.14) RESERVED\n'
  3433 = '(Y102.15) RESERVED\n'
  2494 = '(Y103.00) STN 01 - 05 AGITATION MOTOR ON/OFF (-160K1)'
  7724 = '(Y103.01) LOADING CONVEYOR 01 ON/OFF (-170K1)'
  12715 = '(Y103.02) LOADING CONVEYOR 02 ON/OFF (-171K1)'
  500 = '(Y103.03) LOADING CONVEYOR 03 ON/OFF (-172K1)'
  7713 = '(Y103.04) STATION ROTATION FOR ROTARY BARREL ON/OFF (-4K1 & 2)'
  11682 = '(Y103.05) ROBOT ROTATION FOR ROTARY BARREL ON/OFF (-4K3)'
  155 = '(Y103.06) RESERVED\n'
  13498 = '(Y103.07) RESERVED\n'
  12782 = '(Y103.08) RESERVED\n'
  6048 = '(Y103.09) RESERVED\n'
  1221 = '(Y103.10) RESERVED\n'
  5649 = '(Y103.11) RESERVED\n'
  8397 = '(Y103.12) RESERVED\n'
  8137 = '(Y103.13) RESERVED\n'
  5814 = '(Y103.14) RESERVED\n'
  3911 = '(Y103.15) RESERVED\n'
  6797 = '(Y110.00) STN 03 DOSING PUMP ON/OFF (-72K1)'
  7268 = '(Y110.01) STN 04 DOSING PUMP ON/OFF (-73K1)'
  8036 = '(Y110.02) RESERVED'
  7206 = '(Y110.03) RESERVED'
  10792 = '(Y110.04) RESERVED'
  8398 = '(Y110.05) RESERVED'
  1051 = '(Y110.06) RESERVED'
  9996 = '(Y110.07) RESERVED'
  6956 = '(Y110.08) RESERVED\n'
  4075 = '(Y110.09) RESERVED\n'
  2186 = '(Y110.10) RESERVED\n'
  5827 = '(Y110.11) RESERVED\n'
  271 = '(Y110.12) RESERVED\n'
  3066 = '(Y110.13) RESERVED\n'
  5337 = '(Y110.14) RESERVED\n'
  5157 = '(Y110.15) RESERVED\n'
  9394 = '(Y120.00) STN 01 INCOMING DIW SUPPLY AV1-1 (-420Y1)'
  3345 = '(Y120.01) STN 01 OVERFLOW SUCTION AV1-2 (-420Y2)'
  10197 = '(Y120.02) STN 01 BOTTOM SUCTION AV1-3 (-420Y3)'
  13660 = '(Y120.03) STN 01 DRAIN AV1-4 (-420Y4)'
  14091 = '(Y120.04) STN 02 INCOMING DIW SUPPLY AV2-1 (-420Y5)'
  12279 = '(Y120.05) STN 02 OVERFLOW SUCTION AV2-2 (-420Y6)'
  10215 = '(Y120.06) STN 02 BOTTOM SUCTION AV2-3 (-420Y7)'
  7352 = '(Y120.07) STN 02 DRAIN AV2-4 (-420Y8)'
  3939 = '(Y120.08) STN 03 INCOMING DIW SUPPLY AV3-1 (-420Y9)'
  12053 = '(Y120.09) STN 03 OVERFLOW SUCTION AV3-2 (-420Y10)'
  11532 = '(Y120.10) STN 03 BOTTOM SUCTION AV3-3 (-420Y11)'
  3310 = '(Y120.11) STN 03 DRAIN AV3-4 (-420Y12)'
  2986 = '(Y120.12) STN 04 INCOMING DIW SUPPLY AV4-1 (-420Y13)'
  810 = '(Y120.13) STN 04 OVERFLOW SUCTION AV4-2 (-420Y14)'
  2035 = '(Y120.14) STN 04 BOTTOM SUCTION AV4-3 (-420Y15)'
  6982 = '(Y120.15) STN 04 DRAIN AV4-4 (-420Y16)'
  13694 = '(Y121.00) STN 05 INCOMING DIW SUPPLY AV5-1 (-421Y1)'
  5189 = '(Y121.01) STN 05 OVERFLOW SUCTION AV5-2 (-421Y2)'
  5312 = '(Y121.02) STN 05 BOTTOM SUCTION AV5-3 (-421Y3)'
  7095 = '(Y121.03) STN 05 DRAIN AV5-4 (-421Y4)'
  13007 = '(Y121.04) STN 06 BLOWER PROTECTION AV6-1 (-421Y5)'
  3420 = '(Y121.05) STN 06 BLOWER PROTECTION AV6-2 (-421Y6)'
  1326 = '(Y121.06) STN 06 VACUUM SUCTION AV6-3 (-421Y7)'
  3917 = '(Y121.07) STN 06 VACUUM RELEASE AV6-4 (-421Y8)'
  9590 = '(Y121.08) GENERAL INCOMING DIW SUPPLY AVINC-1 (-421Y9)'
  10324 = '(Y121.09) GENERAL INCOMING CW SUPPLY AVINC-2 (-421Y10)'
  525 = '(Y121.10) RESERVED\n'
  6629 = '(Y121.11) RESERVED\n'
  9736 = '(Y121.12) RESERVED\n'
  5435 = '(Y121.13) RESERVED\n'
  2693 = '(Y121.14) RESERVED\n'
  8606 = '(Y121.15) RESERVED\n'
  14346 = '(Y122.00) STN 06 SHUTTER DOOR - OPEN (-422Y1)'
  10386 = '(Y122.01) STN 06 SHUTTER DOOR - CLOSE (-422Y2)\n'
  7734 = '(Y122.02) STN 06 SHUTTER DOOR - CLAMP (-422Y3)\n'
  11353 = '(Y122.03) STN 06 SHUTTER DOOR - UNCLAMP (-422Y4)\n'
  10729 = '(Y122.04) RESERVED\n'
  13529 = '(Y122.05) RESERVED'
  1773 = '(Y122.06) RESERVED'
  5334 = '(Y122.07) RESERVED\n'
  8088 = '(Y122.08) RESERVED\n'
  5963 = '(Y122.09) RESERVED\n'
  9740 = '(Y122.10) RESERVED\n'
  1559 = '(Y122.11) RESERVED\n'
  2852 = '(Y122.12) RESERVED\n'
  3940 = '(Y122.13) RESERVED\n'
  7536 = '(Y122.14) RESERVED\n'
  4842 = '(Y122.15) RESERVED\n'
  6003 = '1'
  3983 = '10'
  2050 = '11'
  3901 = '12'
  3843 = '13'
  909 = '14'
  1923 = '15'
  4708 = '16'
  2358 = '17'
  2692 = '18'
  2006 = '19'
  10521 = '1ST LIMIT ALARM (+/-)'
  1241 = '1st LIMIT TIMER'
  1993 = '1ST STAGE'
  4717 = '1ST STAGE SPEED PROFILE'
  10596 = '1st VELO (mm/s)'
  5796 = '2'
  1058 = '20'
  4466 = '2nd LIMIT TIMER'
  5210 = '2ND STAGE'
  5091 = '2ND STAGE SPEED PROFILE'
  3977 = '3'
  2859 = '3RD STAGE'
  2965 = '3RD STAGE SPEED PROFILE'
  5216 = '4'
  2573 = '4TH STAGE'
  1367 = '4TH STAGE SPEED PROFILE'
  6822 = '5'
  1400 = '6'
  6329 = '7'
  3152 = '7 DAYS PREPARATION'
  5104 = '8'
  7541 = '9'
  2450 = ':'
  591 = ': %0.01f'
  1846 = 'ACC (mm/s2)'
  1228 = 'ACCESS LEVEL'
  2289 = 'ACTIVE ALARM'
  0 = 'ACTUAL VALUE'
  1966 = 'ADD USER'
  58 = 'ALARM'
  2296 = 'ALARM HISTORY'
  3527 = 'ALARM STATUS'
  658 = 'ARM'
  1473 = 'Arm Busy'
  144 = 'ARM CONTROL'
  502 = 'ARM HOMING :'
  2421 = 'ARM HORIZONTAL HOMING'
  1701 = 'ARM HORIZONTAL POSITION (MM)'
  5912 = 'ARM HORIZONTAL SETTING'
  906 = 'ARM INFO'
  770 = 'ARM JOG VELO (mm/s)'
  21 = 'ARM PATTERN'
  1169 = 'ARM POSITION'
  6108 = 'ARM ROTATION BASKET'
  4587 = 'ARM SPEED PROFILE'
  670 = 'ARM STATUS'
  2861 = 'ARM STN 1 UNHOOK'
  7281 = 'ARM UP'
  2729 = 'ARM UP AND DOWN PATTERN'
  2463 = 'ARM VERTICAL HOMING'
  9150 = 'ARM VERTICAL POSITION (MM)'
  634 = 'ARM VERTICAL SETTING'
  3444 = 'ARM VERTICAL UP'
  365 = 'AUTO\nPREPARATION'
  743 = 'AUTO MODE'
  722 = 'AUTO OPERATION SYSTEM CONTROL'
  911 = 'AUTO ORIGIN'
  1 = 'Auto Pre-Heat'
  1117 = 'AUTO RUN'
  1837 = 'AUTO SHUTDOWN'
  369 = 'AUTO START'
  5376 = 'BAD BASKET TOLERANCE TIME'
  2857 = 'bar'
  3096 = 'Bar'
  310 = 'BARCODE'
  1080 = 'BARCODE\nENABLE'
  1558 = 'BARCODE / QR CODE'
  5575 = 'BARCODE PAGE'
  1313 = 'Barcode Received'
  3624 = 'BARCODE REGISTER'
  344 = 'BARCODE REGISTRATION'
  3053 = 'BARCODE STATUS'
  2682 = 'BASIC'
  3887 = 'BASKET\nQUANTITY'
  6885 = 'BASKET ID'
  773 = 'BASKET QUANTITY'
  3803 = 'BLOWER'
  3646 = 'BOTTOM POSITION'
  2931 = 'BUZZER\nRESET'
  1856 = 'C'
  1434 = 'CALIBRATE DONE'
  3324 = 'CALIBRATE FEED (pulse)'
  285 = 'CALIBRATE IN PROGRESS'
  4915 = 'CALIBRATE RESULT (ml)'
  4390 = 'CALIBRATE START'
  1774 = 'CALIBRATION'
  4131 = 'Cancel'
  2503 = 'CANCEL'
  134 = 'CHANGE PASSWORD'
  2647 = 'CHANGE USER DETAILS AND INFORMATION'
  111 = 'CIRCULATION PUMP'
  6168 = 'CLAMP'
  609 = 'CLEAR'
  6198 = 'CLOSE'
  1340 = 'CONDUCTIVITY'
  943 = 'CONDUCTIVITY (μS)'
  4952 = 'CONFIG'
  1271 = 'CONFIRM'
  791 = 'CONFIRM NEW PASSWORD'
  900 = 'COPY'
  2437 = 'COPY TO\nPROGRAM NO.'
  3155 = 'COPY TO PROGRAM NO.'
  2300 = 'CREATE\nUSER'
  102 = 'CREATE USER ACCOUNT TO GAIN CONTROL ACCESS'
  1958 = 'CURRENT PASSWORD'
  4074 = 'CYCLE'
  852 = 'DAILY'
  691 = 'DAY:HOUR:MIN:SEC'
  873 = 'DCC (mm/s2)'
  493 = 'DEACTIVATED'
  5460 = 'DELETE'
  817 = 'DESCRIPTION'
  3855 = 'DISABLE INSTRUMENT'
  610 = 'DO YOU WANT TO EXIT MANUAL MODE?'
  4016 = 'DOOR'
  6405 = 'DOOR CLAMP'
  4841 = 'DOOR CLOSE'
  2846 = 'DOOR OPEN'
  6495 = 'DOOR STN 6 CLAMP'
  3177 = 'DOOR STN 6 CLOSE'
  6487 = 'DOOR UNCLAMP'
  8544 = 'DOSE PER PULSE (ml)'
  613 = 'DOSING'
  1538 = 'DOSING CALIBRATION'
  2851 = 'DOWN TRANSFER'
  5567 = 'DRIPPING TIME'
  3912 = 'EDIT'
  6373 = 'EDIT AND ADD USER'
  3660 = 'EDIT RECIPE'
  4472 = 'ELAPSED TIME'
  5466 = 'EN'
  7815 = 'ENABLE'
  355 = 'ENGINEER'
  838 = 'ERRORS AND WARNINGS'
  77 = 'EVENT\nRESET'
  815 = 'EVENT ID'
  3463 = 'FILTER'
  767 = 'FILTER PRESSURE (bar)'
  4821 = 'FILTER PRESSURE (Bar)'
  1253 = 'FIRST FILL (ml)'
  1696 = 'FIRST NAME'
  5450 = 'FR'
  6107 = 'FREQ'
  881 = 'FRI , 31MAR 2023 , 9:56:12 AM'
  4621 = 'FRIDAY'
  1542 = 'GENERAL INC CW AVINC-2'
  4155 = 'GENERAL INC DIW AVINC-1'
  7132 = 'GENERAL INC DIW AVINC-2'
  1657 = 'GER'
  3119 = 'HEATER'
  3092 = 'HIGH ALARM'
  203 = 'HIGH SAVE'
  4356 = 'HIGH TEMP ALARM'
  6992 = 'HIGH VACUUM LEVEL'
  2 = 'HOMING SECTION'
  2331 = 'HOOK'
  734 = 'HORIZONTAL'
  2378 = 'HOUR'
  3416 = 'HYSTERESIS'
  253 = 'I/O MONITORING'
  703 = 'ID'
  3523 = 'INCOMING CITY WATER - AV 5-2'
  8167 = 'INCOMING DI WATER - AV 5-1'
  2254 = 'INCOMING VALVE DELAY OFF'
  4371 = 'INPUT'
  330 = 'JOG MODE'
  600 = 'kHz'
  4486 = 'kPa'
  9520 = 'L'
  830 = 'LANGUAGE :'
  599 = 'LAST NAME'
  2728 = 'LD\nDOWN'
  2158 = 'LD\nHOOK'
  1638 = 'LD\nUNHOOK'
  1919 = 'LD CONVEYOR MOTOR 1'
  3077 = 'LD CONVEYOR MOTOR 2'
  3073 = 'LD CONVEYOR MOTOR 3'
  916 = 'LEVEL'
  1155 = 'LIST OF INPUTS AND OUTPUTS'
  1138 = 'LOADING'
  411 = 'LOG IN'
  858 = 'LOG IN TO START OPERATE THE MACHINE'
  1699 = 'Login Name'
  4330 = 'LOW ALARM'
  5373 = 'LOW SAVE'
  1735 = 'LOW VACUUM LEVEL'
  1315 = 'MACHINE INFO'
  191 = 'MACHINE OPERATION HOUR          '
  499 = 'MACHINE VIEW'
  242 = 'MAIN SYSTEM'
  762 = 'MAINTENANCE SYSTEM CONTROL'
  3579 = 'MANUAL BASKET LOAD'
  5048 = 'MANUAL DOSING'
  1580 = 'MANUAL DOSING (ml)'
  468 = 'MANUAL MODE'
  1770 = 'MAXIMUM PROCESS TIME'
  5270 = 'MID POSITION'
  4416 = 'MINIMUM PROCESS TIME'
  460 = 'MINUTE'
  1911 = 'ml'
  4815 = 'MONDAY'
  967 = 'N/A'
  2131 = 'N/A Load Time   :'
  241 = 'NEW PASSWORD'
  1018 = 'NEW USER'
  2698 = 'Next Load Time :'
  5051 = 'NO'
  325 = 'NO.'
  9420 = 'NOTICE !'
  2535 = 'NUMBER OF BASKET\nBETWEEN DOSING'
  816 = 'OCCURRED'
  4569 = 'OFF'
  558 = 'OK'
  4314 = 'ON'
  313 = 'ORIGIN STATUS'
  1211 = 'OTHER INFO'
  7601 = 'OUTPUT'
  1066 = 'OVERVIEW'
  933 = 'PARAMETER'
  1793 = 'PARAMETER\nOVERVIEW'
  6578 = 'PARAMETER OVERVIEW'
  840 = 'PASSWORD'
  1633 = 'PICK & PLACE STATION '
  1474 = 'PICK UP'
  2181 = 'Please key in recipe and press \nthe push button to load the basket'
  2185 = 'POWER'
  267 = 'POWER ON'
  985 = 'PREPARATION STATUS'
  1556 = 'PRESSURE'
  1909 = 'PROCESS'
  363 = 'PROCESS AND HANDLING PRESETS'
  48 = 'PROCESS MANAGEMENT'
  314 = 'PROCESS STATUS'
  3093 = 'PROCESS TANK'
  3650 = 'PROCESS TIME (s)'
  2438 = 'PROCESS TIME SV'
  2980 = 'PRODUCT'
  478 = 'PRODUCT INFO'
  2493 = 'PRODUCT QUALITY'
  2150 = 'PRODUCT RECIPE CONFIGURATION'
  539 = 'PRODUCT RECIPE DESCRIPTION'
  4069 = 'PRODUCT RECIPE NO.'
  772 = 'PV'
  298 = 'QUALITY'
  10625 = 'READY (+/-)'
  57 = 'RECIPE'
  5669 = 'RECIPE DESCRIPTION'
  941 = 'Recipe Name'
  283 = 'RECIPE NAME'
  2788 = 'RECIPE NO'
  571 = 'RECIPE NO.'
  3419 = 'RECIPE OVERVIEW'
  11375 = 'RECIPE PARAMETERS HAVE BEEN SAVED SUCCESSFULLY....'
  564 = 'RECOVERED'
  7121 = 'REFERENCE MAXIMUM VACUUM READING'
  23 = 'REMAINING DOSING\nVOLUME (ml)'
  453 = 'REPEAT FROM\nSTEP NO.'
  1007 = 'RESET'
  1893 = 'Reset'
  281 = 'Reset Done'
  1405 = 'RESET REMAINING\nDOSING TOTALIZER (ml)'
  4071 = 'RESET REMAINING\nDOSING VOLUME (ml)'
  254 = 'RUN'
  5034 = 'SATURDAY'
  53 = 'SAVE'
  667 = 'Scan Complete'
  447 = 'Scan Start'
  4578 = 'SENSOR A MISSHOOK\nALARM DEACTIVATED'
  3015 = 'SENSOR B MISSHOOK\nALARM DEACTIVATED'
  4042 = 'SEQUENCE RECIPE CONFIGURATION (SSER)'
  1305 = 'SEQUENCE RECIPE INFO (SSER)'
  3694 = 'SET TIME'
  1659 = 'SET VALUE'
  197 = 'SETTING'
  669 = 'SLOWPULL'
  4890 = 'SPEED PATTERN NO'
  4281 = 'SPEED PROFILE NO.'
  4424 = 'SSER'
  3904 = 'SSER NAME'
  4062 = 'SSER NO.'
  646 = 'SSUR'
  1459 = 'SSUR NAME'
  1820 = 'SSUR NO.'
  224 = 'START'
  183 = 'STATION'
  370 = 'STATION 01'
  742 = 'STATION 02'
  859 = 'STATION 03'
  200 = 'STATION 04'
  72 = 'STATION 05'
  509 = 'STATION 06'
  4945 = 'STATION 5 INCOMING WATER'
  3 = 'STATION INFO'
  4252 = 'STATION ROTATION\nBASKET'
  2249 = 'STATION VIEW'
  1600 = 'STEP'
  1308 = 'STEP 01'
  541 = 'STEP 02'
  535 = 'STEP 03'
  398 = 'STEP 04'
  1687 = 'STEP 05'
  1286 = 'STEP 06'
  2151 = 'STEP 07'
  1635 = 'STEP 08'
  2165 = 'STEP 09'
  510 = 'STEP 10'
  2122 = 'STEP 11'
  1601 = 'STEP 12'
  1643 = 'STEP 13'
  179 = 'STEP 14'
  2188 = 'STEP 15'
  201 = 'STEP 16'
  1624 = 'STEP 17'
  2332 = 'STEP 18'
  960 = 'STEP 19'
  2078 = 'STEP 20'
  512 = 'STN 01\nDOWN'
  3517 = 'STN 01\nHOOK'
  2972 = 'STN 01\nUNHOOK'
  1354 = 'STN 01 BOTTOM\nSUCTION VALVE AV1-3'
  8043 = 'STN 01 DIW INC\nSUPPLY VALVE AV1-1'
  1834 = 'STN 01 DRAIN\nVALVE AV1-4'
  1064 = 'STN 01 DRAIN \nVALVE AV1-4'
  4000 = 'STN 01 OVERFLOW\nSUCTION VALVE AV1-2'
  1115 = 'STN 01 PROCESS TANK MIN LEVEL'
  1803 = 'STN 01 READY TEMPERATURE'
  2317 = 'STN 02\nDOWN'
  2785 = 'STN 02\nHOOK'
  3442 = 'STN 02\nUNHOOK'
  6777 = 'STN 02 BOTTOM\nSUCTION VALVE AV2-3'
  731 = 'STN 02 DIW INC\nSUPPLY VALVE AV2-1'
  4357 = 'STN 02 DRAIN\nVALVE AV2-4'
  341 = 'STN 02 DRAIN \nVALVE AV2-4'
  3264 = 'STN 02 INC\nSUPPLY VALVE AV2-1'
  6735 = 'STN 02 OVERFLOW\nSUCTION VALVE AV2-2'
  3083 = 'STN 02 OVERFLOW \nSUCTION VALVE AV2-2\n'
  1861 = 'STN 02 PROCESS TANK MIN LEVEL'
  2860 = 'STN 02 READY TEMPERATURE'
  1393 = 'STN 03\nDOWN'
  3367 = 'STN 03\nHOOK'
  4177 = 'STN 03\nUNHOOK'
  4961 = 'STN 03 BOTTOM\nSUCTION VALVE AV3-3'
  8217 = 'STN 03 DIW INC\nSUPPLY VALVE AV3-1'
  4960 = 'STN 03 DRAIN\nVALVE AV3-4'
  1570 = 'STN 03 DRAIN \nVALVE AV3-4'
  979 = 'STN 03 INC\nSUPPLY VALVE AV3-1'
  8087 = 'STN 03 OVERFLOW\nSUCTION VALVE AV3-2'
  7190 = 'STN 03 OVERFLOW \nSUCTION VALVE AV3-2\n'
  949 = 'STN 03 PROCESS TANK MIN LEVEL'
  337 = 'STN 03 READY TEMPERATURE'
  4423 = 'STN 04\nDOWN'
  1019 = 'STN 04\nHOOK'
  2377 = 'STN 04\nUNHOOK'
  4758 = 'STN 04 BOTTOM\nSUCTION VALVE AV4-3'
  6731 = 'STN 04 DIW INC\nSUPPLY VALVE AV4-1'
  6404 = 'STN 04 DRAIN\nVALVE AV4-4'
  6821 = 'STN 04 DRAIN\nVALVE AV5-4'
  2015 = 'STN 04 DRAIN \nVALVE AV4-4'
  1560 = 'STN 04 INC\nSUPPLY VALVE AV4-1'
  2047 = 'STN 04 OVERFLOW\nSUCTION VALVE AV4-2'
  5099 = 'STN 04 OVERFLOW \nSUCTION VALVE AV4-2\n'
  1508 = 'STN 04 PROCESS TANK MIN LEVEL'
  1561 = 'STN 04 READY TEMPERATURE'
  1404 = 'STN 05\nDOWN'
  450 = 'STN 05\nHOOK'
  275 = 'STN 05\nUNHOOK'
  6465 = 'STN 05 BOTTOM\nSUCTION VALVE AV5-3'
  5882 = 'STN 05 DIW INC\nSUPPLY VALVE AV5-1'
  4563 = 'STN 05 DRAIN \nVALVE AV5-4'
  7483 = 'STN 05 INCOMING\nDIW SUPPLY AV5-1'
  8763 = 'STN 05 INCOMING CW \nSUPPLY AV5-2'
  387 = 'STN 05 INCOMING CW \nSUPPLY AV5-2\n'
  986 = 'STN 05 PROCESS TANK MIN LEVEL'
  4491 = 'STN 06\nDOOR CLAMP'
  5348 = 'STN 06\nDOOR CLOSE'
  6314 = 'STN 06\nDOOR OPEN'
  4822 = 'STN 06\nDOOR UNCLAMP'
  2916 = 'STN 06\nDOWN'
  3548 = 'STN 06\nHOOK'
  1817 = 'STN 06\nUNHOOK'
  1963 = 'STN 06 BLOWER \nPROTECTION AV6-1'
  7026 = 'STN 06 BLOWER \nPROTECTION AV6-1\n'
  6675 = 'STN 06 BLOWER \nPROTECTION AV6-2'
  7223 = 'STN 06 BLOWER \nPROTECTION AV6-2\n'
  547 = 'STN 06 READY TEMPERATURE'
  503 = 'STN 06 VACUUM\nRELEASE VALVE AV6-4'
  8004 = 'STN 06 VACUUM\nSUCTION VALVE AV6-3'
  5755 = 'STN 1-4 CHEMICAL RETURN TANK PUMP'
  3161 = 'STN 1-5 AGITATION MOTOR'
  892 = 'STN 1-6 EXHAUST\nBLOWER'
  7438 = 'STN 1-6 EXHAUST BLOWER'
  7765 = 'STN 5-6 FFU UNIT'
  633 = 'STOP'
  664 = 'SUB PROCESS RECIPE CONFIGURATION (SSUR)'
  2224 = 'SUB PROCESS RECIPE INFO (SSUR)'
  1574 = 'SUNDAY'
  2871 = 'SV'
  1513 = 'TAKT TIMER (sec)'
  660 = 'TANK TEMPERATURE (°C)'
  10007 = 'TEMP NOT READY ALARM'
  7215 = 'TEMP PV (°C)  '
  567 = 'TEMPERATURE'
  4669 = 'THURSDAY'
  8390 = 'TIME OPTIMIZE/TRACKER'
  5394 = 'TIMER (sec)'
  1727 = 'TO'
  3738 = 'TOP POSITION'
  222 = 'TOTAL'
  5188 = 'TOTALIZER DOSING\nVOLUME'
  2552 = 'TOTALIZER DOSING\nVOLUME (ml)'
  730 = 'Tracker In progress'
  1022 = 'Tracker Info Available'
  3941 = 'Tracker Info Not Available'
  3628 = 'TUESDAY'
  1934 = 'ULD\nDOWN'
  1088 = 'ULD\nHOOK'
  935 = 'ULD\nUNHOOK'
  2917 = 'ULTRASONIC'
  4066 = 'ULTRASONIC '
  5782 = 'ULTRASONIC BOTTOM'
  1471 = 'ULTRASONIC BOTTOM FREQ (kHz)'
  2017 = 'ULTRASONIC BOTTOM POWER (%)'
  7723 = 'ULTRASONIC FREQ (kHz)'
  2282 = 'ULTRASONIC POWER (%)'
  874 = 'ULTRASONIC SIDE'
  1578 = 'ULTRASONIC SIDE FREQ (kHz)'
  2764 = 'ULTRASONIC SIDE POWER (%)'
  2639 = 'UNHOOK'
  24 = 'UNLOADING'
  2520 = 'UNLOADING BUZZER'
  6626 = 'UNLOADING FFU UNIT'
  459 = 'UP'
  59 = 'USER'
  4288 = 'USER\nSETTING'
  3518 = 'USER LEVEL'
  5968 = 'USER NAME'
  62 = 'USER SETTING'
  8785 = 'VACUUM'
  6841 = 'VACUUM ABOVE TARGET (kPa)'
  6476 = 'VACUUM BELOW TARGET (kPa)'
  4547 = 'VACUUM CALIBRATION'
  4594 = 'VACUUM LEVEL'
  596 = 'VACUUM LEVEL PV '
  6321 = 'VACUUM PRESSURE (bar)'
  6778 = 'VACUUM PUMP'
  5369 = 'VACUUM PUMP MAJOR SERVICE DAYS'
  4691 = 'VACUUM PUMP ROUTINE SERVICE DAYS'
  1822 = 'VACUUM PUMP RUN TIMER'
  1935 = 'VACUUM PUMP SERVICE HOUR'
  2670 = 'VACUUM PUMP SERVICE ROUTINE'
  6275 = 'VACUUM PUMP TIMER'
  7519 = 'VACUUM SYSTEM (kpa)'
  3009 = 'VELOCITY (mm/s)'
  1563 = 'VERTICAL'
  4494 = 'VOLUME PER BASKET (ml)'
  2338 = 'WASHING'
  2654 = 'WEDNESDAY'
  2581 = 'Write Done'
  4553 = 'μS'
END_TEXTLIST

// ---- VISUs/ALARM/Alarm_Page.TcVIS
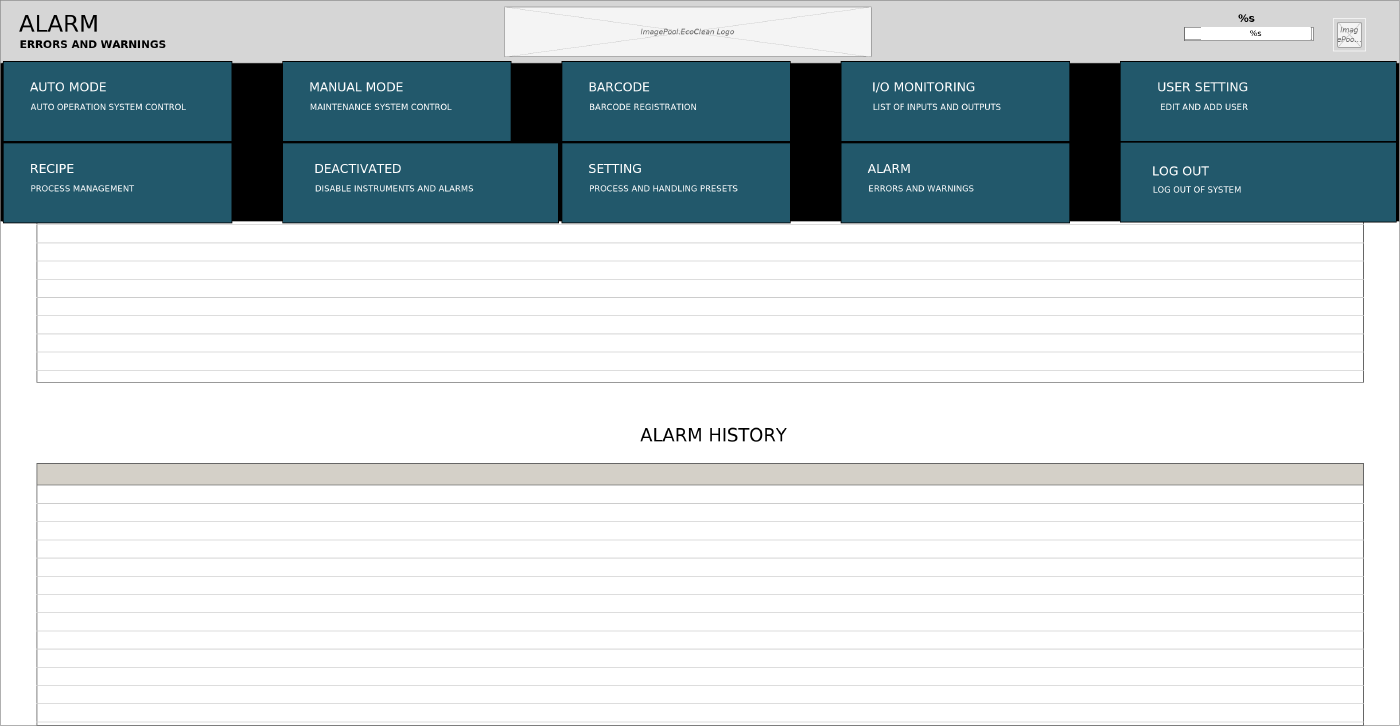
VISUALIZATION Alarm_Page  // 1920x997
    Rectangle (0,63 1920x26)
        p3528305787: HMI_Ctrl.ANIMATION3
    Rectangle (0,0 1919x85)
    Label (23,6 267x53), "ALARM"
    Label (24,49 320x24), "ERRORS AND WARNINGS"
    Group (1828,25 45x45)
        OnMouseClick: toggle HMI_Ctrl.MenuButton
        RoundedRectangle (0,0 45x45), colour toggle: HMI_Ctrl.MenuButton
        Image (6,5 33x35), image: ImagePool.Menu Button
    Rectangle (769,133 419x29), "ACTIVE ALARM"
    Rectangle (769,583 419x29), "ALARM HISTORY"
    Button (1748,119 122x56), "EVENT RESET"
        tap bEventRstPB
    Button (1580,119 122x56), "BUZZER RESET"
        tap bBuzzerRstPB
    Table (50,203 1820x322), data array: ARdsEventActiveDisplay
        p3854506369: ARdsEventActiveDisplay[INDEX].iEventID
        p1892666644: ARdsEventActiveDisplay[INDEX].sTimeAndDate_Occurred
        p338671338: ARdsEventActiveDisplay[INDEX].sEventCode
        p2170511999: ARdsEventActiveDisplay[INDEX].sEventType
        p3723444502: ARdsEventActiveDisplay[INDEX].sLocation
        p1218418051: ARdsEventActiveDisplay[INDEX].sSubLocation
        p746581629: ARdsEventActiveDisplay[INDEX].sDescription
        p3104783080: ARdsEventActiveDisplay[INDEX].sCaused
        p2501879983: ARdsEventActiveDisplay[INDEX].sRemedy
        p2232123230: EVENT ID
        p1791247317: ARdsEventActiveDisplay[INDEX].sEventType_C
    Table (50,636 1820x361), data array: ARdsEventHistoryDisplay
        p3854506369: ARdsEventHistoryDisplay[INDEX].iEventID
        p7306298: ARdsEventHistoryDisplay[INDEX].sCaused
        p1933151965: ARdsEventHistoryDisplay[INDEX].sRemedy
        p1892666644: ARdsEventHistoryDisplay[INDEX].sEventCode
        p511219082: EVENT ID
        p338671338: ARdsEventHistoryDisplay[INDEX].sTimeAndDate_Occurred
        p4092479075: ARdsEventHistoryDisplay[INDEX].sTimeAndDate_Acknowledged
        p2237128397: ARdsEventHistoryDisplay[INDEX].sEventType
        p505689113: ARdsEventHistoryDisplay[INDEX].sLocation
        p1757482276: ARdsEventHistoryDisplay[INDEX].sSubLocation
        p3104783080: ARdsEventHistoryDisplay[INDEX].sDescription
        p2501879983: ARdsEventHistoryDisplay[INDEX].sTimeAndDate_Recovered
    Frame (0,84 1918x221), invisible if: HMI_Ctrl.CloseMenuButton
        shows Popup_MenuPage()
    Image (691,9 504x69), image: ImagePool.EcoClean Logo
    Group (1621,14 180x42)
        Rectangle (0,0 177x22), "%s", text variable: DSLocalSystemTimeML.sCurrentDT24Hr_General
        Button (3,23 177x19), image: VisuSymbols.Symbols.AddUser
        Rectangle (26,23 150x18), "%s", text variable: fbHmiTF1800_UserlevelManagement.dsHmiUserStatus_Active.sLoginName
END_VISUALIZATION

// ---- VISUs/AUTO/AutoMain_Page.TcVIS
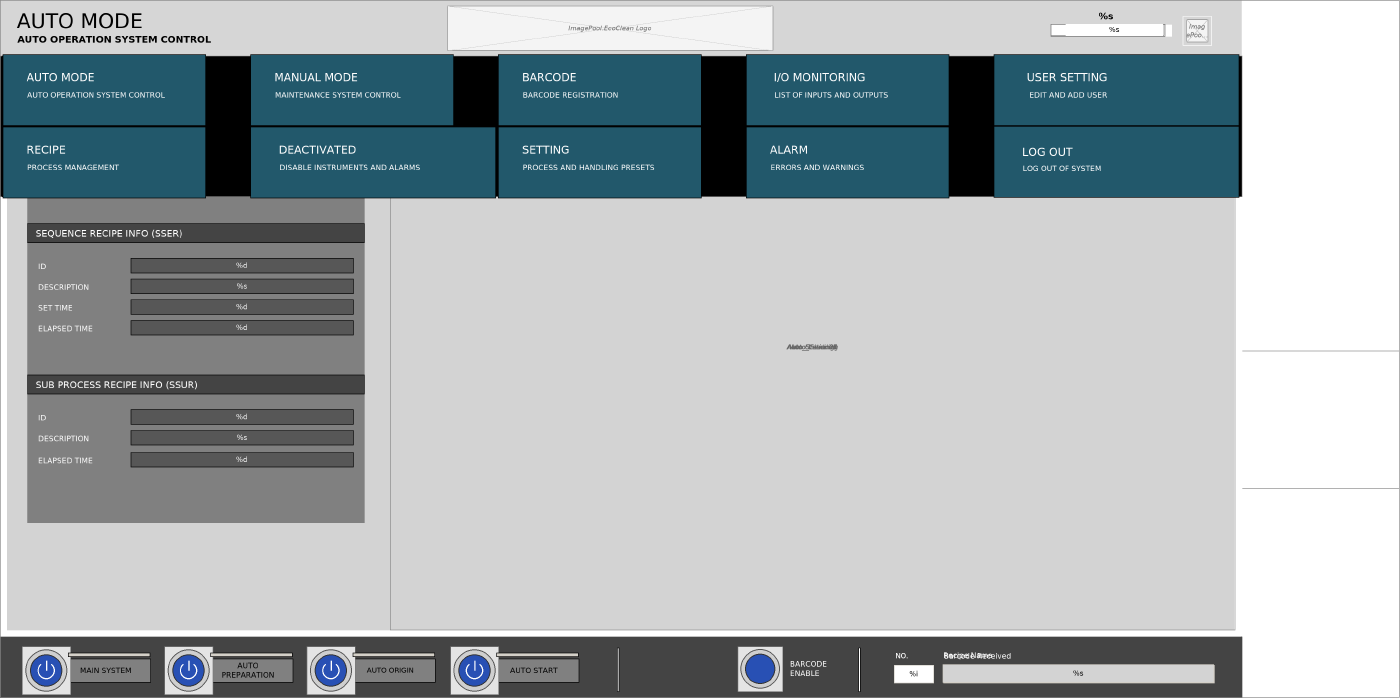
VISUALIZATION AutoMain_Page  // 2164x1079
    Rectangle (0,63 1920x26)
        p3528305787: HMI_Ctrl.ANIMATION3
    Rectangle (0,0 1919x85)
    Label (23,6 267x53), "AUTO MODE"
    Label (24,49 666x24), "AUTO OPERATION SYSTEM CONTROL"
    Frame (2,542 2161x213)
        shows Popup_ProcessStatus()
    Frame (-1,754 1920x240)
        shows Popup_AllInfo()
    Image (1561,275 150x30)
    Frame (64,91 1230x424)
        shows Popup_Machine()
    Group (1828,25 45x45)
        OnMouseClick: toggle HMI_Ctrl.MenuButton
        RoundedRectangle (0,0 45x45), colour toggle: HMI_Ctrl.MenuButton
        Image (6,5 33x35), image: ImagePool.Menu Button
    Group (1604,113 269x41), invisible if: HMI_Ctrl.AutoStationViewEnable
        RoundedRectangle (0,1 269x39)
        Label (1,0 108x41), "MACHINE VIEW"
        Label (161,0 105x41), "STATION VIEW"
        Group (111,6 47x26)
            OnMouseClick: toggle HMI_Ctrl.AutoStationViewEnable
            Group (0,0 47x26)
                Ellipse (0,0 26x26)
                Ellipse (21,0 26x26)
                RoundedRectangle (8,0 29x26)
            Ellipse (1,1 24x24)
            Ellipse (23,1 23x24)
            RoundedRectangle (9,1 28x24)
            Ellipse (5,5 17x17)
    Image (691,9 504x69), image: ImagePool.EcoClean Logo
    Rectangle (1661,38 150x18), "%s", text variable: fbHmiTF1800_UserlevelManagement.dsHmiUserStatus_Active.sLoginName
    Group (1621,14 180x42)
        Rectangle (0,0 177x22), "%s", text variable: DSLocalSystemTimeML.sCurrentDT24Hr_General
        Button (3,23 177x19), image: VisuSymbols.Symbols.AddUser
        Rectangle (26,23 150x18), "%s", text variable: fbHmiTF1800_UserlevelManagement.dsHmiUserStatus_Active.sLoginName
    Frame (340,90 1021x475), invisible if: NOT bParameterPopupPageOn
        shows Popup_Parameter()
    Frame (746,385 486x336), invisible if: NOT bAutoRecipeBarcodeCallPage
        shows Popup_Barcode()
    Button (1732,218 125x54), "PARAMETER OVERVIEW"
        toggle bParameterPopupPageOn
    Frame (0,88 1920x895), invisible if: NOT HMI_Ctrl.AutoStationViewEnable
        shows Auto_AllStation()
    Frame (0,84 1918x221), invisible if: HMI_Ctrl.CloseMenuButton
        shows Popup_MenuPage()
    Rectangle (0,984 1920x95)
    Group (1381,1002 496x54), invisible if: bBarcodeBypass
        Textfield (77,26 419x28), "%s", text variable: sBarcodeScannerReceivedCmd
        Label (0,0 62x24), "NO."
        Label (75,0 418x24), "Barcode Received"
        Textfield (1,26 61x28), "%i", text variable: HMI_Function.iRecipeNoFeed
    PushSwitch (1140,999 70x70), variable: bBarcodeEnable, behaviour: TOGGLE, style: Switch-PushSwitch-Blue
    Label (1218,1017 107x34), "BARCODE ENABLE"
    Rectangle (954,1001 3x68)
    Rectangle (1327,1001 3x68)
    RoundedRectangle (94,1018 139x37), "MAIN SYSTEM"
    PowerSwitch (34,999 75x75), variable: bMainOnOff, behaviour: TOGGLE, style: Switch-PowerSwitch-Blue
    RoundedRectangle (105,1009 127x6), colour toggle: bMainOnOff
    RoundedRectangle (314,1018 139x37), "AUTO PREPARATION"
    PowerSwitch (254,999 75x75), variable: bAutoPreparationPb, behaviour: TOGGLE, style: Switch-PowerSwitch-Blue
    RoundedRectangle (325,1009 127x6), colour toggle: bAutoPreparationDone
    RoundedRectangle (534,1018 139x37), "AUTO ORIGIN"
    PowerSwitch (474,999 75x75), variable: bAutoOriginPb, behaviour: TOGGLE, style: Switch-PowerSwitch-Blue
    RoundedRectangle (545,1009 127x6), colour toggle: bAutoOriginDone
    RoundedRectangle (756,1018 139x37), "AUTO START"
    PowerSwitch (696,999 75x75), variable: bAutoStartPb, behaviour: TOGGLE, style: Switch-PowerSwitch-Blue
    RoundedRectangle (767,1009 127x6), colour toggle: bAutoStartPb
    Group (1381,1001 495x55), invisible if: NOT bBarcodeBypass
        Label (0,1 50x24), "NO."
        Textfield (1,27 61x28), "%i", text variable: iUserDefineProductRecipeNo
            OnMouseDown: write the text variable via VisuDialogs.Numpad
        Textfield (76,26 419x28), "%s", text variable: ARsProductRecipeDescription[iUserDefineProductRecipeNo]
        Label (74,0 417x24), "Recipe Name"
END_VISUALIZATION

// ---- VISUs/AUTO/Auto_AllStation.TcVIS
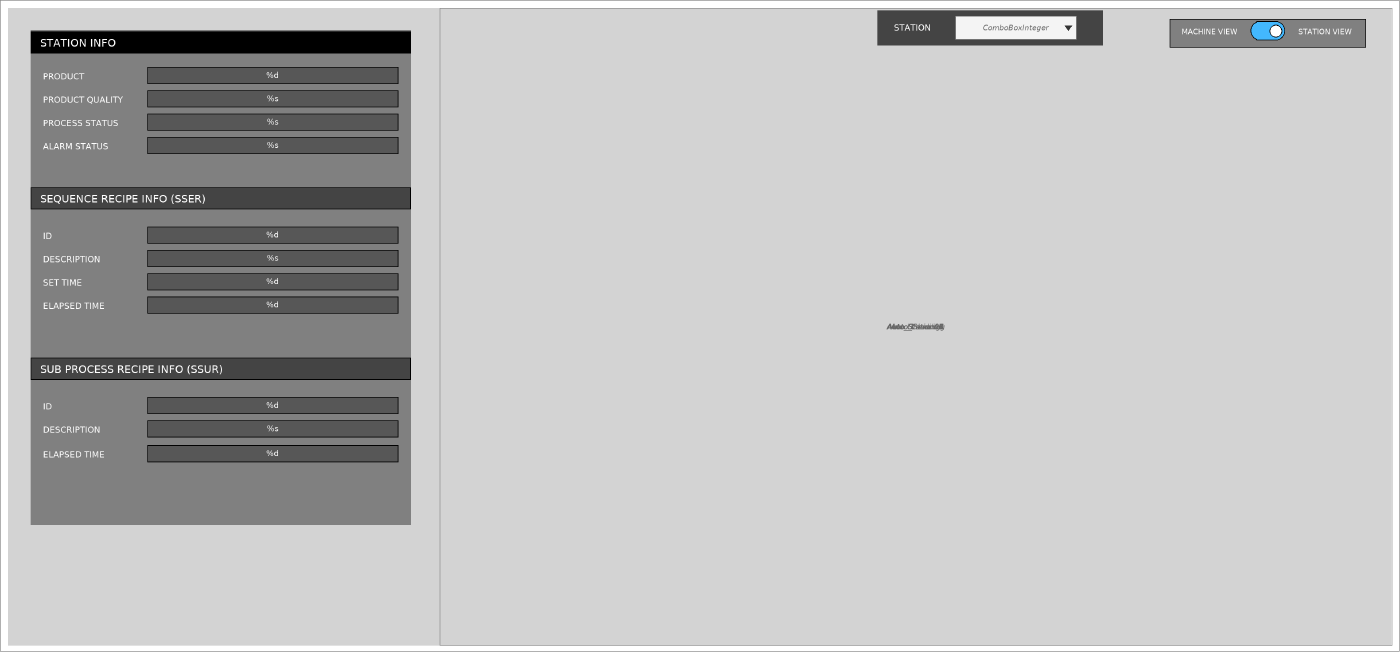
VISUALIZATION Auto_AllStation  // 1920x895
    Rectangle (0,0 1920x895)
    Rectangle (11,11 1896x875)
    Rectangle (42,41 521x679)
    Group (42,43 521x30)
        Rectangle (0,0 521x30)
        Label (10,8 150x16), "STATION INFO"
    Label (56,129 150x16), "PRODUCT QUALITY"
    Rectangle (202,124 344x23), "%s", text variable: DSStnBasketInfo[iAutoStnInfoPageNo].sProductQuality
    Label (56,161 150x16), "PROCESS STATUS"
    Rectangle (202,156 344x23), "%s", text variable: ARsStnProcessStatus[iAutoStnInfoPageNo]
    Label (56,193 150x16), "ALARM STATUS"
    Rectangle (202,188 344x23), "%s", text variable: DSHmiStationDisplayInfo[iAutoStnInfoPageNo].sErrorMessage
    Label (56,412 150x16), "ELAPSED TIME"
    Rectangle (202,407 344x23), "%d", text variable: ARDsStnSeqProcessCtrl[iAutoStnInfoPageNo].Out_iTotalProcessTimeEV
    Label (56,316 150x16), "ID"
    Rectangle (202,311 344x23), "%d", text variable: DSStnBasketInfo[iAutoStnInfoPageNo].iStationSeqenceRecipeNo
    Label (56,348 150x16), "DESCRIPTION"
    Rectangle (202,343 344x23), "%s", text variable: DSHmiStationDisplayInfo[iAutoStnInfoPageNo].sStationSequenceRecipeDescription
    Label (56,380 150x16), "SET TIME"
    Rectangle (202,375 344x23), "%d", text variable: ARDsStnMinMaxEffTimeDisplay[iAutoStnInfoPageNo].iEffTime
    Rectangle (42,257 521x30)
    Label (52,265 496x16), "SEQUENCE RECIPE INFO (SSER)"
    Label (56,616 150x16), "ELAPSED TIME"
    Rectangle (202,611 344x23), "%d", text variable: ARDsStnSeqProcessCtrl[iAutoStnInfoPageNo].Out_iComConProcessTimeEV
    Label (56,550 150x16), "ID"
    Rectangle (202,545 344x23), "%d", text variable: DSStnBasketInfo[iAutoStnInfoPageNo].iProductRecipeStepNo
    Label (56,582 150x16), "DESCRIPTION"
    Rectangle (202,577 344x23), "%s", text variable: DSHmiStationDisplayInfo[iAutoStnInfoPageNo].sStationSubDescription
    Rectangle (42,491 521x30)
    Label (52,499 492x16), "SUB PROCESS RECIPE INFO (SSUR)"
    Rectangle (202,92 344x23), "%d", text variable: DSStnBasketInfo[iAutoStnInfoPageNo].iProductRecipeNo
    Label (56,97 150x16), "PRODUCT"
    Group (603,11 1306x875)
        Frame (0,0 1306x875), invisible if: iAutoStnInfoPageNo <> 2
            shows Auto_Station02()
        Frame (0,0 1306x875), invisible if: iAutoStnInfoPageNo <> 1
            shows Auto_Station01()
        Frame (0,0 1306x875), invisible if: iAutoStnInfoPageNo<> 3
            shows Auto_Station03()
        Frame (0,0 1306x875), invisible if: iAutoStnInfoPageNo <> 4
            shows Auto_Station04()
        Frame (0,0 1306x875), invisible if: iAutoStnInfoPageNo <> 5
            shows Auto_Station05()
        Frame (0,0 1306x875), invisible if: iAutoStnInfoPageNo <> 6
            shows Auto_Station06()
        Frame (0,0 1306x875), invisible if: iAutoStnInfoPageNo <> 7
            shows Auto_Loading()
        Frame (0,0 1306x875), invisible if: iAutoStnInfoPageNo<> 8
            shows Auto_Unloading()
        Frame (0,0 1306x875), invisible if: iAutoStnInfoPageNo<> 9
            shows Auto_General()
    RoundedRectangle (1604,26 269x39)
    Label (1605,23 108x41), "MACHINE VIEW"
    Label (1765,23 105x41), "STATION VIEW"
    Group (1715,29 47x26)
        OnMouseClick: toggle HMI_Ctrl.AutoStationViewEnable
        Group (0,0 47x26)
            Ellipse (0,0 26x26)
            Ellipse (21,0 26x26)
            RoundedRectangle (8,0 29x26)
        Ellipse (1,1 24x24)
        Ellipse (23,1 23x24)
        RoundedRectangle (9,1 28x24)
        Ellipse (26,5 17x17)
    Group (1203,14 288x48)
        RoundedRectangle (0,0 309x48)
        Label (20,12 79x24), "STATION"
    ComboBoxInteger (1310,22 166x32), variable: iAutoStnInfoPageNo, invisible if: NOT HMI_Ctrl.AutoStationViewEnable, text list: 'TextList_SettingPage'
END_VISUALIZATION

// ---- VISUs/BARCODE/Barcode_Page.TcVIS
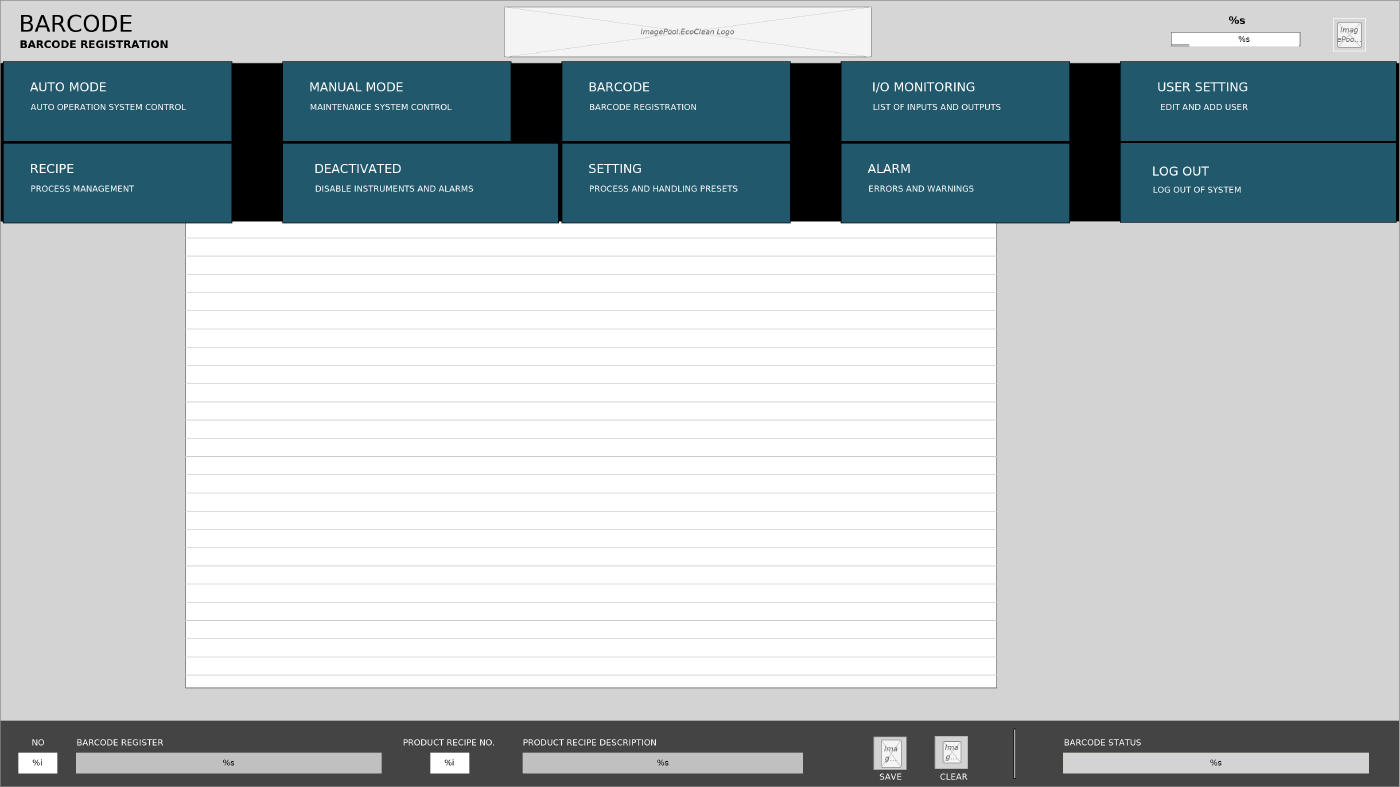
VISUALIZATION Barcode_Page  // 1920x1080
    Rectangle (0,98 1920x981)
    Rectangle (0,63 1920x26)
        p3528305787: HMI_Ctrl.ANIMATION3
    Rectangle (0,0 1919x85)
    Label (23,6 267x53), "BARCODE"
    Label (24,49 320x24), "BARCODE REGISTRATION"
    Rectangle (0,989 1919x91)
    Textfield (1458,1033 419x28), "%s", text variable: Barcode_Reg.sStatus
    Label (1456,1007 127x24), "BARCODE STATUS"
    Rectangle (1390,1000 3x68)
    Textfield (25,1033 53x28), "%i", text variable: iBarcodeRegUserSelectNoDataToSave, input disabled if: iCurrentUserGroupID<3
        OnMouseDown: write the text variable via VisuDialogs.Numpad, min 1, max 100
    Label (26,1007 53x24), "NO"
    Textfield (104,1033 419x28), "%s", text variable: sBarcodeScannerReceivedCmdForReg
    Label (102,1007 413x24), "BARCODE REGISTER"
    Textfield (590,1033 53x28), "%i", text variable: iBarcodeRegUserSelectRecipeNo, input disabled if: iCurrentUserGroupID<3
        OnMouseDown: write the text variable via Default, min 1, max 40
    Label (525,1007 181x24), "PRODUCT RECIPE NO."
    Label (714,1007 387x24), "PRODUCT RECIPE DESCRIPTION"
    Label (1270,1054 76x24), "CLEAR"
    Label (1184,1054 75x24), "SAVE"
    Group (1828,25 45x45)
        OnMouseClick: toggle HMI_Ctrl.MenuButton
        RoundedRectangle (0,0 45x45), colour toggle: HMI_Ctrl.MenuButton
        Image (6,5 33x35), image: ImagePool.Menu Button
    Table (254,196 1113x748), data array: DsAr1sG_BarcodeRegistration
        p3854506369: DsAr1sG_BarcodeRegistration[INDEX].sBarcodeRegistered
        p1892666644: DsAr1sG_BarcodeRegistration[INDEX].iLinkProductRecipeNo
        p338671338: DsAr1sG_BarcodeRegistration[INDEX].bBarcodeRegistrationEn
        p2170511999: DsAr1sG_BarcodeRegistration[INDEX].sLinkProductRecipeDescription
        p2232123230: Barcode Register
        p511219082: Product Recipe
        p4092479075: Product Recipe Description
    Frame (0,84 1918x221), invisible if: HMI_Ctrl.CloseMenuButton
        shows Popup_MenuPage()
    Textfield (717,1033 384x28), "%s", text variable: ARsProductRecipeDescription[iBarcodeRegUserSelectRecipeNo]
    Image (691,9 504x69), image: ImagePool.EcoClean Logo
    Group (1606,17 179x46)
        Button (0,27 177x19), image: VisuSymbols.Symbols.AddUser
        Rectangle (25,28 150x18), "%s", text variable: fbHmiTF1800_UserlevelManagement.dsHmiUserStatus_Active.sLoginName
        Rectangle (2,0 177x22), "%s", text variable: DSLocalSystemTimeML.sCurrentDT24Hr_General
    Group (1198,1011 45x45), input disabled if: bMainOnOff
        RoundedRectangle (0,0 45x45), colour toggle: bBarcodeRegSave
            tap bBarcodeRegSave
        Image (10,4 28x38), image: ImagePool.Save Button
            OnMouseDown: execute { bBarcodeRegSave:=1; }
            OnMouseUp: execute { bBarcodeRegSave:=0; }
    Group (1282,1010 45x45)
        RoundedRectangle (0,0 45x45), colour toggle: bBarcodeRegClear
            tap bBarcodeRegClear
        Image (11,7 25x30), image: ImagePool.Clear Button
            OnMouseDown: execute { bBarcodeRegClear:=1; }
            OnMouseUp: execute { bBarcodeRegClear:=0; }
END_VISUALIZATION

// ---- VISUs/BARCODE/Popup_Barcode.TcVIS
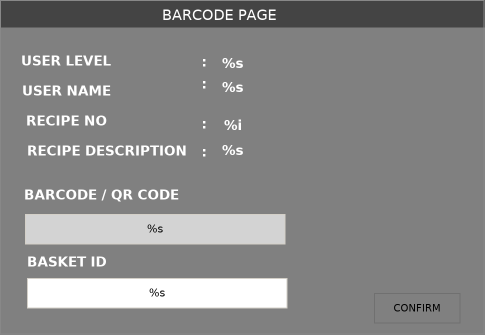
VISUALIZATION Popup_Barcode  // 485x335
    Rectangle (0,0 485x335)
    Rectangle (0,0 485x27)
    Label (159,3 146x24), "BARCODE PAGE"
    Rectangle (219,79 169x17), "%s", text variable: fbHmiTF1800_UserlevelManagement.dsHmiUserReg.ARwsUserGroupName[iLoginNameId]
    Rectangle (219,55 169x17), "%s", text variable: fbHmiTF1800_UserlevelManagement.dsHmiUserReg.ARsLoginName[iLoginNameId]
    Label (18,49 180x24), "USER LEVEL"
    Label (200,57 10x10), ":"
    Label (19,79 179x24), "USER NAME"
    Label (200,79 10x10), ":"
    Label (23,109 177x24), "RECIPE NO"
    Label (200,119 10x10), ":"
    Label (23,139 167x24), "RECIPE DESCRIPTION"
    Label (200,147 10x10), ":"
    Rectangle (221,117 62x17), "%i", text variable: HMI_Function.iRecipeNoFeed
    Rectangle (219,142 169x17), "%s", text variable: ARsProductRecipeDescription[HMI_Function.iRecipeNoFeed]
    Textfield (25,214 260x30), "%s", text variable: sBarcodeScannerReceivedCmd
    Label (21,183 261x24), "BARCODE / QR CODE"
    Button (374,293 86x30), "CONFIRM", colour toggle: bBarcodeConfirm
        tap bBarcodeConfirm
        OnMouseClick: change screen: AutoMain_Page
    Label (24,250 258x24), "BASKET ID"
    Textfield (27,278 260x30), "%s", text variable: sBasketNo
        OnMouseDown: write the text variable via VisuDialogs.Keypad
END_VISUALIZATION

// ---- VISUs/BARCODE/Popup_Ld_Warning.TcVIS
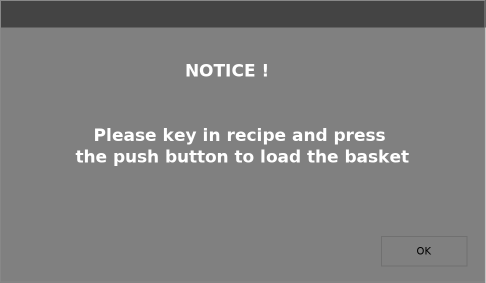
VISUALIZATION Popup_Ld_Warning  // 486x283
    Rectangle (0,0 485x283)
    Rectangle (1,0 485x27)
    Label (152,51 151x39), "NOTICE !"
    Label (10,78 465x136), "Please key in recipe and press the push button to load the basket"
    Button (381,236 86x30), "OK", colour toggle: bPopupPageRapidConfirm
        tap bPopupPageRapidConfirm
END_VISUALIZATION

// ---- VISUs/DEACTIVATED/Deactivated_Page.TcVIS
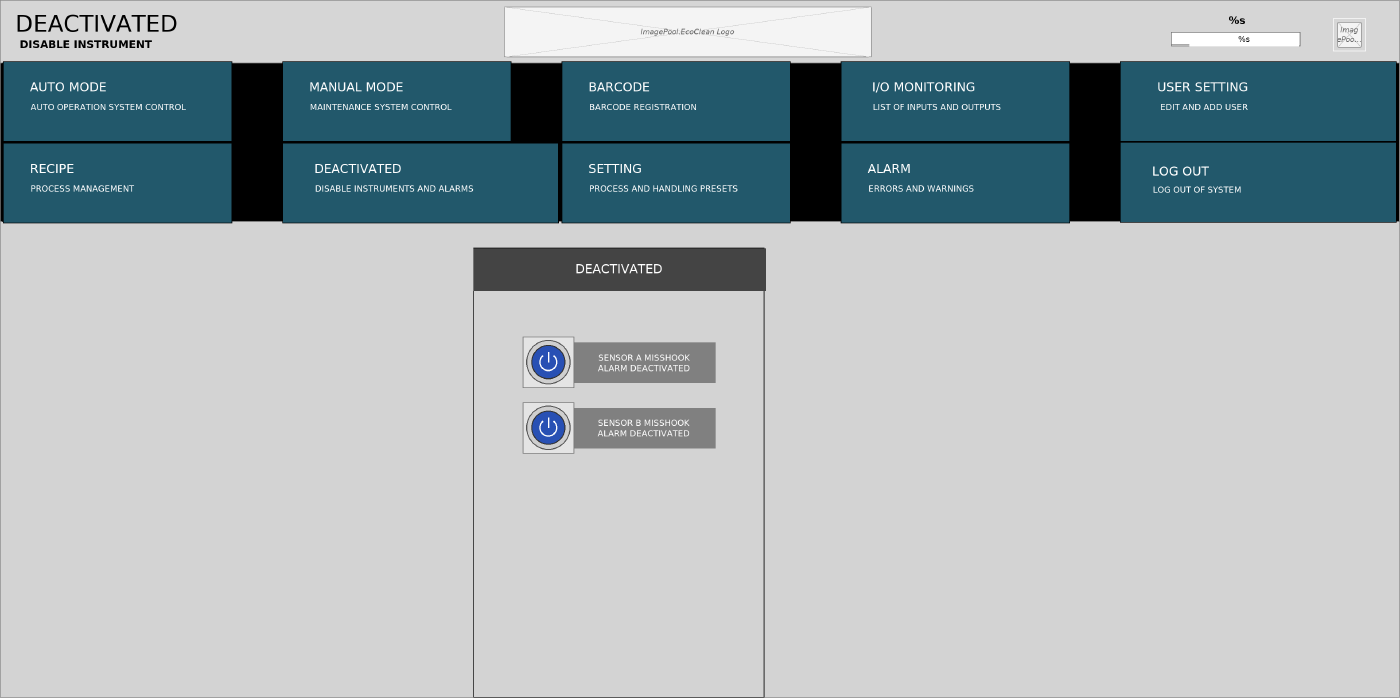
VISUALIZATION Deactivated_Page  // 1920x958
    Rectangle (0,63 1920x26)
        p3528305787: HMI_Ctrl.ANIMATION3
    Rectangle (0,0 1919x85)
    Label (18,6 267x53), "DEACTIVATED"
    Label (24,49 320x24), "DISABLE INSTRUMENT"
    Frame (0,84 1918x221), invisible if: HMI_Ctrl.CloseMenuButton
        shows Popup_MenuPage()
    Group (1828,25 45x45)
        OnMouseClick: toggle HMI_Ctrl.MenuButton
        RoundedRectangle (0,0 45x45), colour toggle: HMI_Ctrl.MenuButton
        Image (6,5 33x35), image: ImagePool.Menu Button
    Rectangle (649,340 399x618)
    Rectangle (649,341 401x58)
    Label (786,357 274x24), "DEACTIVATED"
    RoundedRectangle (766,470 215x55)
    Label (789,473 189x51), "SENSOR A MISSHOOK ALARM DEACTIVATED"
    PowerSwitch (717,462 70x70), variable: ARbArmMissHookByPass1[1], behaviour: TOGGLE, style: Switch-PowerSwitch-Blue
    RoundedRectangle (766,560 215x55)
    Label (788,563 190x50), "SENSOR B MISSHOOK ALARM DEACTIVATED"
    PowerSwitch (717,552 70x70), variable: ARbArmMissHookByPass2[1], behaviour: TOGGLE, style: Switch-PowerSwitch-Blue
    Image (691,9 504x69), image: ImagePool.EcoClean Logo
    Group (1606,17 179x46)
        Button (0,27 177x19), image: VisuSymbols.Symbols.AddUser
        Rectangle (25,28 150x18), "%s", text variable: fbHmiTF1800_UserlevelManagement.dsHmiUserStatus_Active.sLoginName
        Rectangle (2,0 177x22), "%s", text variable: DSLocalSystemTimeML.sCurrentDT24Hr_General
END_VISUALIZATION

